METHOD PROTECTED OnExecute
VAR
    avgStrength : REAL;
END_VAR
hresult.Value := F_VN_LocateAxisAlignedEdges(
    ipSrcImage := ipSrcImage.Value,
    ipEdgePoints := ipEdgePoints.Value,
    aStartPoint := aStartPoint.Value,
    aEndPoint := aEndPoint.Value,
    nSearchWindowHeight := nSearchWindowHeight.Value,
    nKernelSize := nKernelSize.Value,
    nNumEdges := nNumEdges.Value,
    eEdgeSelection := eEdgeSelection.Value,
    fMinStrength := fMinStrength.Value,
    hrPrev := hrPrev.Value,
    fAvgStrength => avgStrength);

fAvgStrength.Value := avgStrength;
END_METHOD

METHOD PUBLIC PreExecutionCheck
VAR_INPUT
    Check : I_PreExecutionChecks;
END_VAR
Check.IsTrue(ipSrcImage.IsValid, 'ipSrcImage must contain an image');
Check.IsTrue(ipSrcImage.HasChannelCount(1), 'ipSrcImage must contain 1 channel');
Check.IsTrue((aStartPoint.Value[0] = aEndPoint.Value[0]) OR (aStartPoint.Value[1] = aEndPoint.Value[1]), 'aEndPoint must share the x- or y-coordinate of aStartPoint');
Check.IsTrue(nSearchWindowHeight.Value > 0, 'nSearchWindowHeight must be at least 1');
Check.IsTrue(nKernelSize.IsOdd, 'nKernelSize must be an odd number');
Check.IsTrue(nKernelSize.Value >= 3, 'nKernelSize must be at least 3');
Check.IsTrue(nNumEdges.Value > 0, 'nNumEdges must be at least 1');
END_METHOD

END_FUNCTION_BLOCK

// Nodes/Measurement/Node_F_VN_LocateAxisAlignedEdgesExp
{attribute 'linkalways'}
{attribute 'no_explicit_call' := 'This FB is a CLASS and must be accessed using methods or properties'}
{attribute 'enable_dynamic_creation'}
FUNCTION_BLOCK Node_F_VN_LocateAxisAlignedEdgesExp EXTENDS VisionNode
VAR
    ipSrcImage : _ITcVnImage;
    ipEdgePoints : _ITcVnContainer;
    aStartPoint : _TcVnPoint2_DINT;
    aEndPoint : _TcVnPoint2_DINT;
    nSearchWindowHeight : _UDINT(1);
    nKernelSize : _UDINT(5);
    nNumEdges : _UDINT(1);
    eEdgeSelection : _ETcVnEdgeSelection(ETcVnEdgeSelection.TCVN_ES_ANY);
    fMinStrength : _REAL(0.0);
    fSigma : _REAL(0.0);
    ipEdgeStrengths : _ITcVnContainer;
    ipDerivative : _ITcVnImage;
    hrPrev : _HRESULT(S_OK);
    fAvgStrength : _REAL(0.0);
    hresult : _HRESULT(S_OK);
END_VAR

METHOD FB_init : BOOL
VAR_INPUT
    bInitRetains : BOOL;
    bInCopyCode : BOOL;
END_VAR
AddInput('ipSrcImage', ipSrcImage);
AddOutput('ipEdgePoints', ipEdgePoints);
AddInput('aStartPoint', aStartPoint);
AddInput('aEndPoint', aEndPoint);
AddParameter('nSearchWindowHeight', nSearchWindowHeight);
AddParameter('nKernelSize', nKernelSize);
AddParameter('nNumEdges', nNumEdges);
AddParameter('eEdgeSelection', eEdgeSelection);
AddParameter('fMinStrength', fMinStrength);
AddParameter('fSigma', fSigma);
AddOutput('ipEdgeStrengths', ipEdgeStrengths);
AddOutput('ipDerivative', ipDerivative);
AddInput('hrPrev', hrPrev);
AddOutput('fAvgStrength', fAvgStrength);
AddOutput('hresult', hresult);
END_METHOD

METHOD PUBLIC Clone : I_Node
VAR
    pNode : POINTER TO Node_F_VN_LocateAxisAlignedEdgesExp;
END_VAR
pNode := __NEW(Node_F_VN_LocateAxisAlignedEdgesExp);
Clone := pNode^;
END_METHOD

METHOD PROTECTED OnExecute
VAR
    avgStrength : REAL;
END_VAR
hresult.Value := F_VN_LocateAxisAlignedEdgesExp(
    ipSrcImage := ipSrcImage.Value,
    ipEdgePoints := ipEdgePoints.Value,
    aStartPoint := aStartPoint.Value,
    aEndPoint := aEndPoint.Value,
    nSearchWindowHeight := nSearchWindowHeight.Value,
    nKernelSize := nKernelSize.Value,
    nNumEdges := nNumEdges.Value,
    eEdgeSelection := eEdgeSelection.Value,
    fMinStrength := fMinStrength.Value,
    fSigma := fSigma.Value,
    ipEdgeStrengths := ipEdgeStrengths.Value,
    ipDerivative := ipDerivative.Value,
    hrPrev := hrPrev.Value,
    fAvgStrength => avgStrength);

fAvgStrength.Value := avgStrength;
END_METHOD

METHOD PUBLIC PreExecutionCheck
VAR_INPUT
    Check : I_PreExecutionChecks;
END_VAR
Check.IsTrue(ipSrcImage.IsValid, 'ipSrcImage must contain an image');
Check.IsTrue(ipSrcImage.HasChannelCount(1), 'ipSrcImage must contain 1 channel');
Check.IsTrue((aStartPoint.Value[0] = aEndPoint.Value[0]) OR (aStartPoint.Value[1] = aEndPoint.Value[1]), 'aEndPoint must share the x- or y-coordinate of aStartPoint');
Check.IsTrue(nSearchWindowHeight.Value > 0, 'nSearchWindowHeight must be at least 1');
Check.IsTrue(nKernelSize.IsOdd, 'nKernelSize must be an odd number');
Check.IsTrue(nKernelSize.Value >= 3, 'nKernelSize must be at least 3');
Check.IsTrue(nNumEdges.Value > 0, 'nNumEdges must be at least 1');
// fSigma = 0 lets the function choose a value from nKernelSize.
Check.IsTrue(fSigma.Value >= 0.0, 'fSigma cannot be negative');
Check.IsTrue((ipDerivative.Value = 0) OR (ipDerivative.Value <> ipSrcImage.Value), 'ipDerivative must be different from the source image');
END_METHOD

END_FUNCTION_BLOCK

// Nodes/Measurement/Node_F_VN_LocateCircularArc
{attribute 'linkalways'} 
{attribute 'no_explicit_call' := 'This FB is a CLASS and must be accessed using methods or properties'}
{attribute 'enable_dynamic_creation'}
FUNCTION_BLOCK Node_F_VN_LocateCircularArc EXTENDS VisionNode
VAR
	ipSrcImage : _ITcVnImage;
	stCircularArc : _TcVnCircularArc;
	aCenter : _TcVnPoint2_REAL;
	fSearchRadius : _REAL(0.0);
	fArcDirectionRad : _LREAL(0.0);
	eEdgeDirection : _ETcVnEdgeDirection(ETcVnEdgeDirection.TCVN_ED_DARK_TO_LIGHT);
    fMinStrength : _REAL(0.0);
	hrPrev : _HRESULT(S_OK);
	hresult : _HRESULT(S_OK);
END_VAR

METHOD FB_init : BOOL
VAR_INPUT
	bInitRetains : BOOL; // if TRUE, the retain variables are initialized (warm start / cold start)
	bInCopyCode : BOOL;  // if TRUE, the instance afterwards gets moved into the copy code (online change)
END_VAR
AddInput('ipSrcImage', ipSrcImage);
AddInput('aCenter', aCenter);
AddInput('hrPrev', hrPrev);
AddParameter('fSearchRadius', fSearchRadius);
AddParameter('fArcDirectionRad', fArcDirectionRad);
AddParameter('eEdgeDirection', eEdgeDirection);
AddParameter('fMinStrength', fMinStrength);
AddOutput('stCircularArc', stCircularArc);
AddOutput('aCenter', aCenter);
AddOutput('hresult',hresult);
END_METHOD

METHOD PUBLIC  Clone : I_Node
VAR
	pNode : POINTER TO Node_F_VN_LocateCircularArc;
END_VAR
pNode := __NEW(Node_F_VN_LocateCircularArc);
Clone := pNode^;
END_METHOD

METHOD PROTECTED OnExecute
hresult.Value := F_VN_LocateCircularArc(
	ipSrcImage := ipSrcImage.Value,
	stCircularArc := stCircularArc.Value,
    aCenter := aCenter.Value,
    fSearchRadius := fSearchRadius.Value,
    fArcDirectionRad := fArcDirectionRad.Value,
	eEdgeDirection := eEdgeDirection.Value,
	fMinStrength := fMinStrength.Value,
	hrPrev := hrPrev.Value);
END_METHOD

METHOD PUBLIC PreExecutionCheck
VAR_INPUT
	Check : I_PreExecutionChecks;
END_VAR
VAR
	width : UDINT;
	height : UDINT;
	cx : REAL;
	cy : REAL;
END_VAR
// Source image (1 channel)
Check.IsTrue(ipSrcImage.IsValid, 'ipSrcImage must contain an image');
Check.IsTrue(ipSrcImage.HasChannelCount(1), 'ipSrcImage must contain 1 channel');
	
// Input search radius (starting FROM aCenter, should be greater than the actual circle radius but 
// aCenter + fSearchRadius should be within the image borders)
ipSrcImage.TryGetWidth(width);
ipSrcImage.TryGetHeight(height);

Check.IsTrue((width > 0), 'ipSrcImage have valid width');
Check.IsTrue((height > 0), 'ipSrcImage have valid height');
Check.IsTrue(fSearchRadius.Value > 0, 'fSearchRadius must be > 0');

cx := aCenter.Value[0];
cy := aCenter.Value[1];

Check.IsTrue(cx - fSearchRadius.Value >= 0, 'Search radius exceeds left border');
Check.IsTrue(cy - fSearchRadius.Value >= 0, 'Search radius exceeds top border');
Check.IsTrue(cx + fSearchRadius.Value < UDINT_TO_REAL(width), 'Search radius exceeds right border');
Check.IsTrue(cy + fSearchRadius.Value < UDINT_TO_REAL(height), 'Search radius exceeds bottom border');

// Input search starting direction in radian. Valid range is [-pi, +pi], where right is 0 rad, 
// top is -pi/2 rad and bottom +pi/2 rad. The circular arc should at least be valid in range 
// fArcDirectionRad +- 0.4 rad.
Check.IsTrue(fArcDirectionRad.Value >= -PI AND fArcDirectionRad.Value <= PI, 'fArcDirectionRad must be in [-pi, +pi]');
Check.IsTrue(fArcDirectionRad.Value - 0.4 >= -PI, 'fArcDirectionRad - 0.4 must be >= -pi');
Check.IsTrue(fArcDirectionRad.Value + 0.4 <=  PI, 'fArcDirectionRad + 0.4 must be <= +pi');
END_METHOD

END_FUNCTION_BLOCK

// Nodes/Measurement/Node_F_VN_LocateCircularArcExp
{attribute 'linkalways'}
{attribute 'no_explicit_call' := 'This FB is a CLASS and must be accessed using methods or properties'}
{attribute 'enable_dynamic_creation'}
FUNCTION_BLOCK Node_F_VN_LocateCircularArcExp EXTENDS VisionNode
VAR
    ipSrcImage : _ITcVnImage;
    stCircularArc : _TcVnCircularArc;
    aCenter : _TcVnPoint2_REAL;
    fSearchRadius : _REAL(0.0);
    fArcDirectionRad : _LREAL(0.0);
    eEdgeDirection : _ETcVnEdgeDirection(ETcVnEdgeDirection.TCVN_ED_DARK_TO_LIGHT);
    fMinStrength : _REAL(0.0);
    fAngleStepRad : _LREAL(0.1);
    nMaxThickness : _UDINT(10);
    bInvertSearchDirection : _BOOL(FALSE);
    nSubpixelsIterations : _UDINT(10);
    fApproxPrecision : _REAL(0.001);
    eAlgorithm : _ETcVnEdgeDetectionAlgorithm(ETcVnEdgeDetectionAlgorithm.TCVN_EDA_INTERPOLATION);
    ipContourPoints : _ITcVnContainer;
    hrPrev : _HRESULT(S_OK);
    hresult : _HRESULT(S_OK);
END_VAR

METHOD FB_init : BOOL
VAR_INPUT
    bInitRetains : BOOL;
    bInCopyCode : BOOL;
END_VAR
AddInput('ipSrcImage', ipSrcImage);
AddOutput('stCircularArc', stCircularArc);
AddInput('aCenter', aCenter);
AddParameter('fSearchRadius', fSearchRadius);
AddParameter('fArcDirectionRad', fArcDirectionRad);
AddParameter('eEdgeDirection', eEdgeDirection);
AddParameter('fMinStrength', fMinStrength);
AddParameter('fAngleStepRad', fAngleStepRad);
AddParameter('nMaxThickness', nMaxThickness);
AddParameter('bInvertSearchDirection', bInvertSearchDirection);
AddParameter('nSubpixelsIterations', nSubpixelsIterations);
AddParameter('fApproxPrecision', fApproxPrecision);
AddParameter('eAlgorithm', eAlgorithm);
AddOutput('ipContourPoints', ipContourPoints);
AddInput('hrPrev', hrPrev);
AddOutput('aCenter', aCenter);
AddOutput('hresult', hresult);
END_METHOD

METHOD PUBLIC Clone : I_Node
VAR
    pNode : POINTER TO Node_F_VN_LocateCircularArcExp;
END_VAR
pNode := __NEW(Node_F_VN_LocateCircularArcExp);
Clone := pNode^;
END_METHOD

METHOD PROTECTED OnExecute
hresult.Value := F_VN_LocateCircularArcExp(
    ipSrcImage := ipSrcImage.Value,
    stCircularArc := stCircularArc.Value,
    aCenter := aCenter.Value,
    fSearchRadius := fSearchRadius.Value,
    fArcDirectionRad := fArcDirectionRad.Value,
    eEdgeDirection := eEdgeDirection.Value,
    fMinStrength := fMinStrength.Value,
    fAngleStepRad := fAngleStepRad.Value,
    nMaxThickness := nMaxThickness.Value,
    bInvertSearchDirection := bInvertSearchDirection.Value,
    nSubpixelsIterations := nSubpixelsIterations.Value,
    fApproxPrecision := fApproxPrecision.Value,
    eAlgorithm := eAlgorithm.Value,
    ipContourPoints := ipContourPoints.Value,
    hrPrev := hrPrev.Value);
END_METHOD

METHOD PUBLIC PreExecutionCheck
VAR_INPUT
    Check : I_PreExecutionChecks;
END_VAR
VAR
    width : UDINT;
    height : UDINT;
    cx : REAL;
    cy : REAL;
END_VAR
Check.IsTrue(ipSrcImage.IsValid, 'ipSrcImage must contain an image');
Check.IsTrue(ipSrcImage.HasChannelCount(1), 'ipSrcImage must contain 1 channel');

// Input search radius (starting FROM aCenter, should be greater than the actual radius but
// aCenter + fSearchRadius should be within the image borders)
ipSrcImage.TryGetWidth(width);
ipSrcImage.TryGetHeight(height);

Check.IsTrue((width > 0), 'ipSrcImage have valid width');
Check.IsTrue((height > 0), 'ipSrcImage have valid height');
Check.IsTrue(fSearchRadius.Value > 0, 'fSearchRadius must be > 0');

cx := aCenter.Value[0];
cy := aCenter.Value[1];

Check.IsTrue(cx - fSearchRadius.Value >= 0, 'Search radius exceeds left border');
Check.IsTrue(cy - fSearchRadius.Value >= 0, 'Search radius exceeds top border');
Check.IsTrue(cx + fSearchRadius.Value < UDINT_TO_REAL(width), 'Search radius exceeds right border');
Check.IsTrue(cy + fSearchRadius.Value < UDINT_TO_REAL(height), 'Search radius exceeds bottom border');

// Input search starting direction in radian. Valid range is [-pi, +pi], where right is 0 rad,
// top is -pi/2 rad and bottom +pi/2 rad. The circular arc should at least be valid in range
// fArcDirectionRad +- 4 * fAngleStepRad.
Check.IsTrue(fAngleStepRad.Value > 0.0, 'fAngleStepRad must be greater than 0');
Check.IsTrue(fArcDirectionRad.Value >= -PI AND fArcDirectionRad.Value <= PI, 'fArcDirectionRad must be in [-pi, +pi]');
Check.IsTrue(fArcDirectionRad.Value - 4.0 * fAngleStepRad.Value >= -PI, 'fArcDirectionRad - 4 * fAngleStepRad must be >= -pi');
Check.IsTrue(fArcDirectionRad.Value + 4.0 * fAngleStepRad.Value <=  PI, 'fArcDirectionRad + 4 * fAngleStepRad must be <= +pi');

Check.IsTrue(nMaxThickness.Value > 0, 'nMaxThickness must be at least 1');
Check.IsTrue(nSubpixelsIterations.Value > 0, 'nSubpixelsIterations must be greater than 0');
Check.IsTrue((eAlgorithm.Value = ETcVnEdgeDetectionAlgorithm.TCVN_EDA_INTERPOLATION) OR
             (fApproxPrecision.Value > 0.0), 'fApproxPrecision must be greater than 0 for the approximation algorithms');
END_METHOD

END_FUNCTION_BLOCK

// Nodes/Measurement/Node_F_VN_LocateCircularArcExp2
{attribute 'linkalways'}
{attribute 'no_explicit_call' := 'This FB is a CLASS and must be accessed using methods or properties'}
{attribute 'enable_dynamic_creation'}
FUNCTION_BLOCK Node_F_VN_LocateCircularArcExp2 EXTENDS VisionNode
VAR
    ipSrcImage : _ITcVnImage;
    stCircularArc : _TcVnCircularArc;
    aCenter : _TcVnPoint2_REAL;
    fSearchRadius : _REAL(0.0);
    fArcDirectionRad : _LREAL(0.0);
    eEdgeDirection : _ETcVnEdgeDirection(ETcVnEdgeDirection.TCVN_ED_DARK_TO_LIGHT);
    fMinStrength : _REAL(0.0);
    fAngleStepRad : _LREAL(0.1);
    nMaxThickness : _UDINT(10);
    bInvertSearchDirection : _BOOL(FALSE);
    nSubpixelsIterations : _UDINT(10);
    fApproxPrecision : _REAL(0.001);
    eAlgorithm : _ETcVnEdgeDetectionAlgorithm(ETcVnEdgeDetectionAlgorithm.TCVN_EDA_INTERPOLATION);
    ipContourPoints : _ITcVnContainer;
    fRangeCutoffFactor : _REAL(0.135);
    hrPrev : _HRESULT(S_OK);
    hresult : _HRESULT(S_OK);
END_VAR

METHOD FB_init : BOOL
VAR_INPUT
    bInitRetains : BOOL;
    bInCopyCode : BOOL;
END_VAR
AddInput('ipSrcImage', ipSrcImage);
AddOutput('stCircularArc', stCircularArc);
AddInput('aCenter', aCenter);
AddParameter('fSearchRadius', fSearchRadius);
AddParameter('fArcDirectionRad', fArcDirectionRad);
AddParameter('eEdgeDirection', eEdgeDirection);
AddParameter('fMinStrength', fMinStrength);
AddParameter('fAngleStepRad', fAngleStepRad);
AddParameter('nMaxThickness', nMaxThickness);
AddParameter('bInvertSearchDirection', bInvertSearchDirection);
AddParameter('nSubpixelsIterations', nSubpixelsIterations);
AddParameter('fApproxPrecision', fApproxPrecision);
AddParameter('eAlgorithm', eAlgorithm);
AddOutput('ipContourPoints', ipContourPoints);
AddParameter('fRangeCutoffFactor', fRangeCutoffFactor);
AddInput('hrPrev', hrPrev);
AddOutput('aCenter', aCenter);
AddOutput('hresult', hresult);
END_METHOD

METHOD PUBLIC Clone : I_Node
VAR
    pNode : POINTER TO Node_F_VN_LocateCircularArcExp2;
END_VAR
pNode := __NEW(Node_F_VN_LocateCircularArcExp2);
Clone := pNode^;
END_METHOD

METHOD PROTECTED OnExecute
hresult.Value := F_VN_LocateCircularArcExp2(
    ipSrcImage := ipSrcImage.Value,
    stCircularArc := stCircularArc.Value,
    aCenter := aCenter.Value,
    fSearchRadius := fSearchRadius.Value,
    fArcDirectionRad := fArcDirectionRad.Value,
    eEdgeDirection := eEdgeDirection.Value,
    fMinStrength := fMinStrength.Value,
    fAngleStepRad := fAngleStepRad.Value,
    nMaxThickness := nMaxThickness.Value,
    bInvertSearchDirection := bInvertSearchDirection.Value,
    nSubpixelsIterations := nSubpixelsIterations.Value,
    fApproxPrecision := fApproxPrecision.Value,
    eAlgorithm := eAlgorithm.Value,
    ipContourPoints := ipContourPoints.Value,
    fRangeCutoffFactor := fRangeCutoffFactor.Value,
    hrPrev := hrPrev.Value);
END_METHOD

METHOD PUBLIC PreExecutionCheck
VAR_INPUT
    Check : I_PreExecutionChecks;
END_VAR
VAR
    width : UDINT;
    height : UDINT;
    cx : REAL;
    cy : REAL;
END_VAR
Check.IsTrue(ipSrcImage.IsValid, 'ipSrcImage must contain an image');
Check.IsTrue(ipSrcImage.HasChannelCount(1), 'ipSrcImage must contain 1 channel');

// Input search radius (starting FROM aCenter, should be greater than the actual radius but
// aCenter + fSearchRadius should be within the image borders)
ipSrcImage.TryGetWidth(width);
ipSrcImage.TryGetHeight(height);

Check.IsTrue((width > 0), 'ipSrcImage have valid width');
Check.IsTrue((height > 0), 'ipSrcImage have valid height');
Check.IsTrue(fSearchRadius.Value > 0, 'fSearchRadius must be > 0');

cx := aCenter.Value[0];
cy := aCenter.Value[1];

Check.IsTrue(cx - fSearchRadius.Value >= 0, 'Search radius exceeds left border');
Check.IsTrue(cy - fSearchRadius.Value >= 0, 'Search radius exceeds top border');
Check.IsTrue(cx + fSearchRadius.Value < UDINT_TO_REAL(width), 'Search radius exceeds right border');
Check.IsTrue(cy + fSearchRadius.Value < UDINT_TO_REAL(height), 'Search radius exceeds bottom border');

// Input search starting direction in radian. Valid range is [-pi, +pi], where right is 0 rad,
// top is -pi/2 rad and bottom +pi/2 rad. The circular arc should at least be valid in range
// fArcDirectionRad +- 4 * fAngleStepRad.
Check.IsTrue(fAngleStepRad.Value > 0.0, 'fAngleStepRad must be greater than 0');
Check.IsTrue(fArcDirectionRad.Value >= -PI AND fArcDirectionRad.Value <= PI, 'fArcDirectionRad must be in [-pi, +pi]');
Check.IsTrue(fArcDirectionRad.Value - 4.0 * fAngleStepRad.Value >= -PI, 'fArcDirectionRad - 4 * fAngleStepRad must be >= -pi');
Check.IsTrue(fArcDirectionRad.Value + 4.0 * fAngleStepRad.Value <=  PI, 'fArcDirectionRad + 4 * fAngleStepRad must be <= +pi');

Check.IsTrue(nMaxThickness.Value > 0, 'nMaxThickness must be at least 1');
Check.IsTrue(nSubpixelsIterations.Value > 0, 'nSubpixelsIterations must be greater than 0');
Check.IsTrue((eAlgorithm.Value = ETcVnEdgeDetectionAlgorithm.TCVN_EDA_INTERPOLATION) OR
             (fApproxPrecision.Value > 0.0), 'fApproxPrecision must be greater than 0 for the approximation algorithms');
END_METHOD

END_FUNCTION_BLOCK

// Nodes/Measurement/Node_F_VN_LocateEdge
{attribute 'linkalways'} 
{attribute 'no_explicit_call' := 'This FB is a CLASS and must be accessed using methods or properties'}
{attribute 'enable_dynamic_creation'}
FUNCTION_BLOCK Node_F_VN_LocateEdge EXTENDS VisionNode
VAR
	ipSrcImage : _ITcVnImage;
    ipEdgePoints : _ITcVnContainer;
    aStartPoint : _TcVnPoint2_REAL;
    aEndPoint : _TcVnPoint2_REAL;
	eEdgeDirection : _ETcVnEdgeDirection(ETcVnEdgeDirection.TCVN_ED_DARK_TO_LIGHT);
    fMinStrength : _REAL(0.0);
    nSearchLines : _UDINT(1);
    hrPrev : _HRESULT(S_OK);
    fAvgStrength : _REAL(0.0);
	hresult : _HRESULT(S_OK);
END_VAR

METHOD FB_init : BOOL
VAR_INPUT
	bInitRetains : BOOL; // if TRUE, the retain variables are initialized (warm start / cold start)
	bInCopyCode : BOOL;  // if TRUE, the instance afterwards gets moved into the copy code (online change)
END_VAR
AddInput('ipSrcImage', ipSrcImage);
AddInput('aStartPoint', aStartPoint);
AddInput('aEndPoint', aEndPoint);
AddParameter('eEdgeDirection', eEdgeDirection);
AddParameter('fMinStrength', fMinStrength);
AddParameter('nSearchLines', nSearchLines);
AddInput('hrPrev', hrPrev);
AddOutput('ipEdgePoints', ipEdgePoints);
AddOutput('fAvgStrength', fAvgStrength);
AddOutput('hresult',hresult);
END_METHOD

METHOD PUBLIC  Clone : I_Node
VAR
	pNode : POINTER TO Node_F_VN_LocateEdge;
END_VAR
pNode := __NEW(Node_F_VN_LocateEdge);
Clone := pNode^;
END_METHOD

METHOD PROTECTED OnExecute
VAR
    avgStrength : REAL;
END_VAR
hresult.Value := F_VN_LocateEdge(
	ipSrcImage := ipSrcImage.Value,
	ipEdgePoints := ipEdgePoints.Value,
    aStartPoint := aStartPoint.Value,
    aEndPoint := aEndPoint.Value,
    eEdgeDirection := eEdgeDirection.Value,
	fMinStrength := fMinStrength.Value,
	nSearchLines := nSearchLines.Value,
	hrPrev := hrPrev.Value,
    fAvgStrength => avgStrength);
    
fAvgStrength.Value := avgStrength;
END_METHOD

METHOD PUBLIC PreExecutionCheck
VAR_INPUT
	Check : I_PreExecutionChecks;
END_VAR
Check.IsTrue(ipSrcImage.IsValid, 'ipSrcImage must contain an image');
Check.IsTrue(ipSrcImage.HasChannelCount(1), 'ipSrcImage must contain 1 channel');
Check.IsTrue(nSearchLines.IsOdd, 'nSearchLines must be an odd number');
END_METHOD

END_FUNCTION_BLOCK

// Nodes/Measurement/Node_F_VN_LocateEdgeExp
{attribute 'linkalways'} 
{attribute 'no_explicit_call' := 'This FB is a CLASS and must be accessed using methods or properties'}
{attribute 'enable_dynamic_creation'}
FUNCTION_BLOCK Node_F_VN_LocateEdgeExp EXTENDS VisionNode
VAR
	ipSrcImage : _ITcVnImage;
    ipEdgePoints : _ITcVnContainer;
    aStartPoint : _TcVnPoint2_REAL;
    aEndPoint : _TcVnPoint2_REAL;
	eEdgeDirection : _ETcVnEdgeDirection(ETcVnEdgeDirection.TCVN_ED_DARK_TO_LIGHT);
    fMinStrength : _REAL(0.0);
    nSearchLines : _UDINT(1);
    fSearchLineDist : _REAL(0.0);
    nMaxThickness : _UDINT(0);
    nSubpixelsIterations : _UDINT(0);
    fApproxPrecision : _REAL(0.0);
    eAlgorithm : _ETcVnEdgeDetectionAlgorithm(ETcVnEdgeDetectionAlgorithm.TCVN_EDA_INTERPOLATION);
    hrPrev : _HRESULT(S_OK);
    fAvgStrength : _REAL(0.0);
	hresult : _HRESULT(S_OK);
END_VAR

METHOD FB_init : BOOL
VAR_INPUT
	bInitRetains : BOOL; // if TRUE, the retain variables are initialized (warm start / cold start)
	bInCopyCode : BOOL;  // if TRUE, the instance afterwards gets moved into the copy code (online change)
END_VAR
AddInput('ipSrcImage', ipSrcImage);
AddInput('aStartPoint', aStartPoint);
AddInput('aEndPoint', aEndPoint);
AddParameter('eEdgeDirection', eEdgeDirection);
AddParameter('fMinStrength', fMinStrength);
AddParameter('nSearchLines', nSearchLines);
AddParameter('fSearchLineDist', fSearchLineDist);
AddParameter('nMaxThickness', nMaxThickness);
AddParameter('nSubpixelsIterations', nSubpixelsIterations);
AddParameter('fApproxPrecision', fApproxPrecision);
AddParameter('eAlgorithm', eAlgorithm);
AddInput('hrPrev', hrPrev);
AddOutput('ipEdgePoints', ipEdgePoints);
AddOutput('fAvgStrength', fAvgStrength);
AddOutput('hresult',hresult);
END_METHOD

METHOD PUBLIC  Clone : I_Node
VAR
	pNode : POINTER TO Node_F_VN_LocateEdgeExp;
END_VAR
pNode := __NEW(Node_F_VN_LocateEdgeExp);
Clone := pNode^;
END_METHOD

METHOD PROTECTED OnExecute
VAR
    avgStrength : REAL;
END_VAR
hresult.Value := F_VN_LocateEdgeExp(
	ipSrcImage := ipSrcImage.Value,
	ipEdgePoints := ipEdgePoints.Value,
    aStartPoint := aStartPoint.Value,
    aEndPoint := aEndPoint.Value,
    eEdgeDirection := eEdgeDirection.Value,
	fMinStrength := fMinStrength.Value,
	nSearchLines := nSearchLines.Value,
    fSearchLineDist := fSearchLineDist.Value,
    nMaxThickness := nMaxThickness.Value,
    nSubpixelsIterations := nSubpixelsIterations.Value,
    fApproxPrecision := fApproxPrecision.Value,
    eAlgorithm := eAlgorithm.Value,
	hrPrev:= hrPrev.Value,
    fAvgStrength => avgStrength);
    
fAvgStrength.Value := avgStrength;
END_METHOD

METHOD PUBLIC PreExecutionCheck
VAR_INPUT
	Check : I_PreExecutionChecks;
END_VAR
Check.IsTrue(ipSrcImage.IsValid, 'ipSrcImage must contain an image');
Check.IsTrue(ipSrcImage.HasChannelCount(1), 'ipSrcImage must contain 1 channel');
Check.IsTrue(nSearchLines.IsOdd, 'nSearchLines must be an odd number');
Check.IsTrue((fSearchLineDist.Value > 0.0), 'nSearchLineDist must be greater than 0');
END_METHOD

END_FUNCTION_BLOCK

// Nodes/Measurement/Node_F_VN_LocateEdgeExp2
{attribute 'linkalways'}
{attribute 'no_explicit_call' := 'This FB is a CLASS and must be accessed using methods or properties'}
{attribute 'enable_dynamic_creation'}
FUNCTION_BLOCK Node_F_VN_LocateEdgeExp2 EXTENDS VisionNode
VAR
    ipSrcImage : _ITcVnImage;
    ipEdgePoints : _ITcVnContainer;
    aStartPoint : _TcVnPoint2_REAL;
    aEndPoint : _TcVnPoint2_REAL;
    eEdgeDirection : _ETcVnEdgeDirection(ETcVnEdgeDirection.TCVN_ED_DARK_TO_LIGHT);
    fMinStrength : _REAL(0.0);
    nSearchLines : _UDINT(1);
    fSearchLineDist : _REAL(1.0);
    nMaxThickness : _UDINT(10);
    nSubpixelsIterations : _UDINT(10);
    fApproxPrecision : _REAL(0.001);
    eAlgorithm : _ETcVnEdgeDetectionAlgorithm(ETcVnEdgeDetectionAlgorithm.TCVN_EDA_INTERPOLATION);
    fRangeCutoffFactor : _REAL(0.135);
    ipEdgeStrengths : _ITcVnContainer;
    hrPrev : _HRESULT(S_OK);
    fAvgStrength : _REAL(0.0);
    hresult : _HRESULT(S_OK);
END_VAR

METHOD FB_init : BOOL
VAR_INPUT
    bInitRetains : BOOL;
    bInCopyCode : BOOL;
END_VAR
AddInput('ipSrcImage', ipSrcImage);
AddOutput('ipEdgePoints', ipEdgePoints);
AddInput('aStartPoint', aStartPoint);
AddInput('aEndPoint', aEndPoint);
AddParameter('eEdgeDirection', eEdgeDirection);
AddParameter('fMinStrength', fMinStrength);
AddParameter('nSearchLines', nSearchLines);
AddParameter('fSearchLineDist', fSearchLineDist);
AddParameter('nMaxThickness', nMaxThickness);
AddParameter('nSubpixelsIterations', nSubpixelsIterations);
AddParameter('fApproxPrecision', fApproxPrecision);
AddParameter('eAlgorithm', eAlgorithm);
AddParameter('fRangeCutoffFactor', fRangeCutoffFactor);
AddOutput('ipEdgeStrengths', ipEdgeStrengths);
AddInput('hrPrev', hrPrev);
AddOutput('fAvgStrength', fAvgStrength);
AddOutput('hresult', hresult);
END_METHOD

METHOD PUBLIC Clone : I_Node
VAR
    pNode : POINTER TO Node_F_VN_LocateEdgeExp2;
END_VAR
pNode := __NEW(Node_F_VN_LocateEdgeExp2);
Clone := pNode^;
END_METHOD

METHOD PROTECTED OnExecute
VAR
    avgStrength : REAL;
END_VAR
hresult.Value := F_VN_LocateEdgeExp2(
    ipSrcImage := ipSrcImage.Value,
    ipEdgePoints := ipEdgePoints.Value,
    aStartPoint := aStartPoint.Value,
    aEndPoint := aEndPoint.Value,
    eEdgeDirection := eEdgeDirection.Value,
    fMinStrength := fMinStrength.Value,
    nSearchLines := nSearchLines.Value,
    fSearchLineDist := fSearchLineDist.Value,
    nMaxThickness := nMaxThickness.Value,
    nSubpixelsIterations := nSubpixelsIterations.Value,
    fApproxPrecision := fApproxPrecision.Value,
    eAlgorithm := eAlgorithm.Value,
    fRangeCutoffFactor := fRangeCutoffFactor.Value,
    ipEdgeStrengths := ipEdgeStrengths.Value,
    hrPrev := hrPrev.Value,
    fAvgStrength => avgStrength);

fAvgStrength.Value := avgStrength;
END_METHOD

METHOD PUBLIC PreExecutionCheck
VAR_INPUT
    Check : I_PreExecutionChecks;
END_VAR
Check.IsTrue(ipSrcImage.IsValid, 'ipSrcImage must contain an image');
Check.IsTrue(ipSrcImage.HasChannelCount(1), 'ipSrcImage must contain 1 channel');
Check.IsTrue(nSearchLines.IsOdd, 'nSearchLines must be an odd number');
Check.IsTrue(fSearchLineDist.Value > 0.0, 'fSearchLineDist must be greater than 0');
Check.IsTrue(nMaxThickness.Value > 0, 'nMaxThickness must be at least 1');
Check.IsTrue(nSubpixelsIterations.Value > 0, 'nSubpixelsIterations must be greater than 0');
Check.IsTrue((eAlgorithm.Value = ETcVnEdgeDetectionAlgorithm.TCVN_EDA_INTERPOLATION) OR
             (fApproxPrecision.Value > 0.0), 'fApproxPrecision must be greater than 0 for the approximation algorithms');
END_METHOD

END_FUNCTION_BLOCK

// Nodes/Measurement/Node_F_VN_LocateEdges
{attribute 'linkalways'} 
{attribute 'no_explicit_call' := 'This FB is a CLASS and must be accessed using methods or properties'}
{attribute 'enable_dynamic_creation'}
FUNCTION_BLOCK Node_F_VN_LocateEdges EXTENDS VisionNode
VAR
	ipSrcImage : _ITcVnImage;
    ipEdgePoints : _ITcVnContainer;
    aStartPoint : _TcVnPoint2_REAL;
    aEndPoint : _TcVnPoint2_REAL;
    nNumEdges : _UDINT(0);
	eEdgeDirection : _ETcVnEdgeDirection(ETcVnEdgeDirection.TCVN_ED_DARK_TO_LIGHT);
    bAlternateDirection : _BOOL(FALSE);
    fMinStrength : _REAL(0.0);
    nSearchLines : _UDINT(1);
    hrPrev : _HRESULT(S_OK);
    fAvgStrength : _REAL(0.0);
	hresult : _HRESULT(S_OK);
END_VAR

METHOD FB_init : BOOL
VAR_INPUT
	bInitRetains : BOOL; // if TRUE, the retain variables are initialized (warm start / cold start)
	bInCopyCode : BOOL;  // if TRUE, the instance afterwards gets moved into the copy code (online change)
END_VAR
AddInput('ipSrcImage', ipSrcImage);
AddInput('aStartPoint', aStartPoint);
AddInput('aEndPoint', aEndPoint);
AddParameter('nNumEdges', nNumEdges);
AddParameter('eEdgeDirection', eEdgeDirection);
AddParameter('bAlternateDirection', bAlternateDirection);
AddParameter('fMinStrength', fMinStrength);
AddParameter('nSearchLines', nSearchLines);
AddInput('hrPrev', hrPrev);
AddOutput('ipEdgePoints', ipEdgePoints);
AddOutput('fAvgStrength', fAvgStrength);
AddOutput('hresult',hresult);
END_METHOD

METHOD PUBLIC  Clone : I_Node
VAR
	pNode : POINTER TO Node_F_VN_LocateEdges;
END_VAR
pNode := __NEW(Node_F_VN_LocateEdges);
Clone := pNode^;
END_METHOD

METHOD PROTECTED OnExecute
VAR
    avgStrength : REAL;
END_VAR
hresult.Value := F_VN_LocateEdges(
	ipSrcImage := ipSrcImage.Value,
	ipEdgePoints := ipEdgePoints.Value,
    aStartPoint := aStartPoint.Value,
    aEndPoint := aEndPoint.Value,
    nNumEdges := nNumEdges.Value,
    eEdgeDirection := eEdgeDirection.Value,
    bAlternateDirection := bAlternateDirection.Value,
	fMinStrength := fMinStrength.Value,
	nSearchLines := nSearchLines.Value,
	hrPrev := hrPrev.Value,
    fAvgStrength => avgStrength);
    
fAvgStrength.Value := avgStrength;
END_METHOD

METHOD PUBLIC PreExecutionCheck
VAR_INPUT
	Check : I_PreExecutionChecks;
END_VAR
Check.IsTrue(ipSrcImage.IsValid, 'ipSrcImage must contain an image');
Check.IsTrue(ipSrcImage.HasChannelCount(1), 'ipSrcImage must contain 1 channel');
Check.IsTrue(nSearchLines.IsOdd, 'nSearchLines must be an odd number');
END_METHOD

END_FUNCTION_BLOCK

// Nodes/Measurement/Node_F_VN_LocateEdgesExp
{attribute 'linkalways'} 
{attribute 'no_explicit_call' := 'This FB is a CLASS and must be accessed using methods or properties'}
{attribute 'enable_dynamic_creation'}
FUNCTION_BLOCK Node_F_VN_LocateEdgesExp EXTENDS VisionNode
VAR
	ipSrcImage : _ITcVnImage;
    ipEdgePoints : _ITcVnContainer;
    aStartPoint : _TcVnPoint2_REAL;
    aEndPoint : _TcVnPoint2_REAL;
    nNumEdges : _UDINT(0);
	eEdgeDirection : _ETcVnEdgeDirection(ETcVnEdgeDirection.TCVN_ED_DARK_TO_LIGHT);
    bAlternateDirection : _BOOL(FALSE);
    fMinStrength : _REAL(0.0);
    nSearchLines : _UDINT(1);
    fSearchLineDist : _REAL(0.0);
    nMaxThickness : _UDINT(0);
    nSubpixelsIterations : _UDINT(0);
    fApproxPrecision : _REAL(0.0);
    eAlgorithm : _ETcVnEdgeDetectionAlgorithm(ETcVnEdgeDetectionAlgorithm.TCVN_EDA_INTERPOLATION);
    hrPrev : _HRESULT(S_OK);
    fAvgStrength : _REAL(0.0);
	hresult : _HRESULT(S_OK);
END_VAR

METHOD FB_init : BOOL
VAR_INPUT
	bInitRetains : BOOL; // if TRUE, the retain variables are initialized (warm start / cold start)
	bInCopyCode : BOOL;  // if TRUE, the instance afterwards gets moved into the copy code (online change)
END_VAR
AddInput('ipSrcImage', ipSrcImage);
AddInput('aStartPoint', aStartPoint);
AddInput('aEndPoint', aEndPoint);
AddParameter('nNumEdges', nNumEdges);
AddParameter('eEdgeDirection', eEdgeDirection);
AddParameter('bAlternateDirection', bAlternateDirection);
AddParameter('fMinStrength', fMinStrength);
AddParameter('nSearchLines', nSearchLines);
AddParameter('fSearchLineDist', fSearchLineDist);
AddParameter('nMaxThickness', nMaxThickness);
AddParameter('nSubpixelsIterations', nSubpixelsIterations);
AddParameter('fApproxPrecision', fApproxPrecision);
AddParameter('eAlgorithm', eAlgorithm);
AddInput('hrPrev', hrPrev);
AddOutput('ipEdgePoints', ipEdgePoints);
AddOutput('fAvgStrength', fAvgStrength);
AddOutput('hresult',hresult);
END_METHOD

METHOD PUBLIC  Clone : I_Node
VAR
	pNode : POINTER TO Node_F_VN_LocateEdgesExp;
END_VAR
pNode := __NEW(Node_F_VN_LocateEdgesExp);
Clone := pNode^;
END_METHOD

METHOD PROTECTED OnExecute
VAR
    avgStrength : REAL;
END_VAR
hresult.Value := F_VN_LocateEdgesExp(
	ipSrcImage := ipSrcImage.Value,
	ipEdgePoints := ipEdgePoints.Value,
    aStartPoint := aStartPoint.Value,
    aEndPoint := aEndPoint.Value,
    nNumEdges := nNumEdges.Value,
    eEdgeDirection := eEdgeDirection.Value,
    bAlternateDirection := bAlternateDirection.Value,
	fMinStrength := fMinStrength.Value,
	nSearchLines := nSearchLines.Value,
    fSearchLineDist := fSearchLineDist.Value,
    nMaxThickness := nMaxThickness.Value,
    nSubpixelsIterations := nSubpixelsIterations.Value,
    fApproxPrecision := fApproxPrecision.Value,
    eAlgorithm := eAlgorithm.Value,
	hrPrev := hrPrev.Value,
    fAvgStrength => avgStrength);
    
fAvgStrength.Value := avgStrength;
END_METHOD

METHOD PUBLIC PreExecutionCheck
VAR_INPUT
	Check : I_PreExecutionChecks;
END_VAR
Check.IsTrue(ipSrcImage.IsValid, 'ipSrcImage must contain an image');
Check.IsTrue(ipSrcImage.HasChannelCount(1), 'ipSrcImage must contain 1 channel');
Check.IsTrue(nSearchLines.IsOdd, 'nSearchLines must be an odd number');
Check.IsTrue((fSearchLineDist.Value > 0.0), 'nSearchLineDist must be greater than 0');
END_METHOD

END_FUNCTION_BLOCK

// Nodes/Measurement/Node_F_VN_LocateEdgesExp2
{attribute 'linkalways'}
{attribute 'no_explicit_call' := 'This FB is a CLASS and must be accessed using methods or properties'}
{attribute 'enable_dynamic_creation'}
FUNCTION_BLOCK Node_F_VN_LocateEdgesExp2 EXTENDS VisionNode
VAR
    ipSrcImage : _ITcVnImage;
    ipEdgePoints : _ITcVnContainer;
    aStartPoint : _TcVnPoint2_REAL;
    aEndPoint : _TcVnPoint2_REAL;
    nNumEdges : _UDINT(1);
    eEdgeDirection : _ETcVnEdgeDirection(ETcVnEdgeDirection.TCVN_ED_DARK_TO_LIGHT);
    bAlternateDirection : _BOOL(FALSE);
    fMinStrength : _REAL(0.0);
    nSearchLines : _UDINT(1);
    fSearchLineDist : _REAL(1.0);
    nMaxThickness : _UDINT(10);
    nSubpixelsIterations : _UDINT(10);
    fApproxPrecision : _REAL(0.001);
    eAlgorithm : _ETcVnEdgeDetectionAlgorithm(ETcVnEdgeDetectionAlgorithm.TCVN_EDA_INTERPOLATION);
    fRangeCutoffFactor : _REAL(0.135);
    ipEdgeStrengths : _ITcVnContainer;
    bAvgEdgeStrengths : _BOOL(FALSE);
    hrPrev : _HRESULT(S_OK);
    fAvgStrength : _REAL(0.0);
    hresult : _HRESULT(S_OK);
END_VAR

METHOD FB_init : BOOL
VAR_INPUT
    bInitRetains : BOOL;
    bInCopyCode : BOOL;
END_VAR
AddInput('ipSrcImage', ipSrcImage);
AddOutput('ipEdgePoints', ipEdgePoints);
AddInput('aStartPoint', aStartPoint);
AddInput('aEndPoint', aEndPoint);
AddParameter('nNumEdges', nNumEdges);
AddParameter('eEdgeDirection', eEdgeDirection);
AddParameter('bAlternateDirection', bAlternateDirection);
AddParameter('fMinStrength', fMinStrength);
AddParameter('nSearchLines', nSearchLines);
AddParameter('fSearchLineDist', fSearchLineDist);
AddParameter('nMaxThickness', nMaxThickness);
AddParameter('nSubpixelsIterations', nSubpixelsIterations);
AddParameter('fApproxPrecision', fApproxPrecision);
AddParameter('eAlgorithm', eAlgorithm);
AddParameter('fRangeCutoffFactor', fRangeCutoffFactor);
AddOutput('ipEdgeStrengths', ipEdgeStrengths);
AddParameter('bAvgEdgeStrengths', bAvgEdgeStrengths);
AddInput('hrPrev', hrPrev);
AddOutput('fAvgStrength', fAvgStrength);
AddOutput('hresult', hresult);
END_METHOD

METHOD PUBLIC Clone : I_Node
VAR
    pNode : POINTER TO Node_F_VN_LocateEdgesExp2;
END_VAR
pNode := __NEW(Node_F_VN_LocateEdgesExp2);
Clone := pNode^;
END_METHOD

METHOD PROTECTED OnExecute
VAR
    avgStrength : REAL;
END_VAR
hresult.Value := F_VN_LocateEdgesExp2(
    ipSrcImage := ipSrcImage.Value,
    ipEdgePoints := ipEdgePoints.Value,
    aStartPoint := aStartPoint.Value,
    aEndPoint := aEndPoint.Value,
    nNumEdges := nNumEdges.Value,
    eEdgeDirection := eEdgeDirection.Value,
    bAlternateDirection := bAlternateDirection.Value,
    fMinStrength := fMinStrength.Value,
    nSearchLines := nSearchLines.Value,
    fSearchLineDist := fSearchLineDist.Value,
    nMaxThickness := nMaxThickness.Value,
    nSubpixelsIterations := nSubpixelsIterations.Value,
    fApproxPrecision := fApproxPrecision.Value,
    eAlgorithm := eAlgorithm.Value,
    fRangeCutoffFactor := fRangeCutoffFactor.Value,
    ipEdgeStrengths := ipEdgeStrengths.Value,
    bAvgEdgeStrengths := bAvgEdgeStrengths.Value,
    hrPrev := hrPrev.Value,
    fAvgStrength => avgStrength);

fAvgStrength.Value := avgStrength;
END_METHOD

METHOD PUBLIC PreExecutionCheck
VAR_INPUT
    Check : I_PreExecutionChecks;
END_VAR
Check.IsTrue(ipSrcImage.IsValid, 'ipSrcImage must contain an image');
Check.IsTrue(ipSrcImage.HasChannelCount(1), 'ipSrcImage must contain 1 channel');
Check.IsTrue(nNumEdges.Value > 0, 'nNumEdges must be at least 1');
Check.IsTrue(nSearchLines.IsOdd, 'nSearchLines must be an odd number');
Check.IsTrue(fSearchLineDist.Value > 0.0, 'fSearchLineDist must be greater than 0');
Check.IsTrue(nMaxThickness.Value > 0, 'nMaxThickness must be at least 1');
Check.IsTrue(nSubpixelsIterations.Value > 0, 'nSubpixelsIterations must be greater than 0');
Check.IsTrue((eAlgorithm.Value = ETcVnEdgeDetectionAlgorithm.TCVN_EDA_INTERPOLATION) OR
             (fApproxPrecision.Value > 0.0), 'fApproxPrecision must be greater than 0 for the approximation algorithms');
END_METHOD

END_FUNCTION_BLOCK

// Nodes/Measurement/Node_F_VN_LocateEllipse
{attribute 'linkalways'} 
{attribute 'no_explicit_call' := 'This FB is a CLASS and must be accessed using methods or properties'}
{attribute 'enable_dynamic_creation'}
FUNCTION_BLOCK Node_F_VN_LocateEllipse EXTENDS VisionNode
VAR
	ipSrcImage : _ITcVnImage;
    stEllipse : _TcVnRotatedRectangle;
    aCenter : _TcVnPoint2_REAL;
    fSearchRadius : _REAL(0.0);
	eEdgeDirection : _ETcVnEdgeDirection(ETcVnEdgeDirection.TCVN_ED_DARK_TO_LIGHT);
    fMinStrength : _REAL(0.0);
    hrPrev : _HRESULT(S_OK);
	hresult : _HRESULT(S_OK);
END_VAR

METHOD FB_init : BOOL
VAR_INPUT
	bInitRetains : BOOL; // if TRUE, the retain variables are initialized (warm start / cold start)
	bInCopyCode : BOOL;  // if TRUE, the instance afterwards gets moved into the copy code (online change)
END_VAR
AddInput('ipSrcImage', ipSrcImage);
AddInput('aCenter', aCenter);
AddParameter('fSearchRadius', fSearchRadius);
AddParameter('eEdgeDirection', eEdgeDirection);
AddParameter('fMinStrength', fMinStrength);
AddInput('hrPrev', hrPrev);
AddOutput('stEllipse', stEllipse);
AddOutput('hresult',hresult);
END_METHOD

METHOD PUBLIC  Clone : I_Node
VAR
	pNode : POINTER TO Node_F_VN_LocateEllipse;
END_VAR
pNode := __NEW(Node_F_VN_LocateEllipse);
Clone := pNode^;
END_METHOD

METHOD PROTECTED OnExecute
hresult.Value := F_VN_LocateEllipse(
	ipSrcImage := ipSrcImage.Value,
    stEllipse := stEllipse.Value,
    aCenter := aCenter.Value,
    fSearchRadius := fSearchRadius.Value,
    eEdgeDirection := eEdgeDirection.Value,
	fMinStrength := fMinStrength.Value,
	hrPrev:= hrPrev.Value);
END_METHOD

METHOD PUBLIC PreExecutionCheck
VAR_INPUT
	Check : I_PreExecutionChecks;
END_VAR
Check.IsTrue(ipSrcImage.IsValid, 'ipSrcImage must contain an image');
Check.IsTrue(ipSrcImage.HasChannelCount(1), 'ipSrcImage must contain 1 channel');
END_METHOD

END_FUNCTION_BLOCK

// Nodes/Measurement/Node_F_VN_LocateEllipseExp
{attribute 'linkalways'} 
{attribute 'no_explicit_call' := 'This FB is a CLASS and must be accessed using methods or properties'}
{attribute 'enable_dynamic_creation'}
FUNCTION_BLOCK Node_F_VN_LocateEllipseExp EXTENDS VisionNode
VAR
	ipSrcImage : _ITcVnImage;
    stEllipse : _TcVnRotatedRectangle;
    aCenter : _TcVnPoint2_REAL;
    fSearchRadius : _REAL(0.0);
	eEdgeDirection : _ETcVnEdgeDirection(ETcVnEdgeDirection.TCVN_ED_DARK_TO_LIGHT);
    fMinStrength : _REAL(0.0);
	nMaxThickness : _UDINT(1);
	fMinSearchRadius : _REAL(0.0);
	bInvertSearchDirection : _BOOL(FALSE);
	nSubpixelsIterations : _UDINT(10);
	nSearchLines : _UDINT(1);
	fApproxPrecision : _REAL(0.001);
	eAlgorithm : _ETcVnEdgeDetectionAlgorithm(ETcVnEdgeDetectionAlgorithm.TCVN_EDA_APPROX_ERF);
	ipContourPoints : _ITcVnContainer;
    hrPrev : _HRESULT(S_OK);
	hresult : _HRESULT(S_OK);
END_VAR

METHOD FB_init : BOOL
VAR_INPUT
	bInitRetains : BOOL; // if TRUE, the retain variables are initialized (warm start / cold start)
	bInCopyCode : BOOL;  // if TRUE, the instance afterwards gets moved into the copy code (online change)
END_VAR
AddInput('ipSrcImage', ipSrcImage);
AddInput('aCenter', aCenter);
AddInput('hrPrev', hrPrev);
AddParameter('fSearchRadius', fSearchRadius);
AddParameter('eEdgeDirection', eEdgeDirection);
AddParameter('fMinStrength', fMinStrength);
AddParameter('nMaxThickness', nMaxThickness);
AddParameter('bInvertSearchDirection', bInvertSearchDirection);
AddParameter('fMinSearchRadius', fMinSearchRadius);
AddParameter('nSubpixelsIterations', nSubpixelsIterations);
AddParameter('nSearchLines', nSearchLines);
AddParameter('fApproxPrecision', fApproxPrecision);
AddParameter('eAlgorithm', eAlgorithm);
AddOutput('stEllipse', stEllipse);
AddOutput('aCenter', aCenter);
AddOutput('ipContourPoints', ipContourPoints);
AddOutput('hresult',hresult);
END_METHOD

METHOD PUBLIC  Clone : I_Node
VAR
	pNode : POINTER TO Node_F_VN_LocateEllipseExp;
END_VAR
pNode := __NEW(Node_F_VN_LocateEllipseExp);
Clone := pNode^;
END_METHOD

METHOD PROTECTED OnExecute
hresult.Value := F_VN_LocateEllipseExp(
	ipSrcImage := ipSrcImage.Value,
    stEllipse := stEllipse.Value,
    aCenter := aCenter.Value,
    fSearchRadius := fSearchRadius.Value,
    eEdgeDirection := eEdgeDirection.Value,
	fMinStrength := fMinStrength.Value,
	nMaxThickness := nMaxThickness.Value,
	bInvertSearchDirection := bInvertSearchDirection.Value,
	fMinSearchRadius := fMinSearchRadius.Value,
	nSubpixelsIterations := nSubpixelsIterations.Value,
	nSearchLines := nSearchLines.Value,
	fApproxPrecision := fApproxPrecision.Value,
	eAlgorithm := eAlgorithm.Value,
	ipContourPoints := ipContourPoints.Value,
	hrPrev:= hrPrev.Value);
END_METHOD

METHOD PUBLIC PreExecutionCheck
VAR_INPUT
	Check : I_PreExecutionChecks;
END_VAR
Check.IsTrue(ipSrcImage.IsValid, 'ipSrcImage must contain an image');
Check.IsTrue(ipSrcImage.HasChannelCount(1), 'ipSrcImage must contain 1 channel');

// Specifies the amount of search lines, which are equally distributed in all directions (must be >= 8 and a multiple of 4)
Check.IsTrue(nSearchLines.Value >= 8, 'nSearchLines must be >= 8');
Check.IsTrue(nSearchLines.Value MOD 4 = 0, 'nSearchLines must be a multiple of 4');
END_METHOD

END_FUNCTION_BLOCK

// Nodes/Measurement/Node_F_VN_LocateEllipseExp2
{attribute 'linkalways'}
{attribute 'no_explicit_call' := 'This FB is a CLASS and must be accessed using methods or properties'}
{attribute 'enable_dynamic_creation'}
FUNCTION_BLOCK Node_F_VN_LocateEllipseExp2 EXTENDS VisionNode
VAR
    ipSrcImage : _ITcVnImage;
    stEllipse : _TcVnRotatedRectangle;
    aCenter : _TcVnPoint2_REAL;
    fSearchRadius : _REAL(0.0);
    eEdgeDirection : _ETcVnEdgeDirection(ETcVnEdgeDirection.TCVN_ED_DARK_TO_LIGHT);
    fMinStrength : _REAL(0.0);
    nMaxThickness : _UDINT(10);
    bInvertSearchDirection : _BOOL(FALSE);
    fMinSearchRadius : _REAL(0.0);
    nSubpixelsIterations : _UDINT(10);
    nSearchLines : _UDINT(92);
    fApproxPrecision : _REAL(0.001);
    eAlgorithm : _ETcVnEdgeDetectionAlgorithm(ETcVnEdgeDetectionAlgorithm.TCVN_EDA_INTERPOLATION);
    ipContourPoints : _ITcVnContainer;
    fRangeCutoffFactor : _REAL(0.135);
    hrPrev : _HRESULT(S_OK);
    hresult : _HRESULT(S_OK);
END_VAR

METHOD FB_init : BOOL
VAR_INPUT
    bInitRetains : BOOL;
    bInCopyCode : BOOL;
END_VAR
AddInput('ipSrcImage', ipSrcImage);
AddOutput('stEllipse', stEllipse);
AddInput('aCenter', aCenter);
AddParameter('fSearchRadius', fSearchRadius);
AddParameter('eEdgeDirection', eEdgeDirection);
AddParameter('fMinStrength', fMinStrength);
AddParameter('nMaxThickness', nMaxThickness);
AddParameter('bInvertSearchDirection', bInvertSearchDirection);
AddParameter('fMinSearchRadius', fMinSearchRadius);
AddParameter('nSubpixelsIterations', nSubpixelsIterations);
AddParameter('nSearchLines', nSearchLines);
AddParameter('fApproxPrecision', fApproxPrecision);
AddParameter('eAlgorithm', eAlgorithm);
AddOutput('ipContourPoints', ipContourPoints);
AddParameter('fRangeCutoffFactor', fRangeCutoffFactor);
AddInput('hrPrev', hrPrev);
AddOutput('aCenter', aCenter);
AddOutput('hresult', hresult);
END_METHOD

METHOD PUBLIC Clone : I_Node
VAR
    pNode : POINTER TO Node_F_VN_LocateEllipseExp2;
END_VAR
pNode := __NEW(Node_F_VN_LocateEllipseExp2);
Clone := pNode^;
END_METHOD

METHOD PROTECTED OnExecute
hresult.Value := F_VN_LocateEllipseExp2(
    ipSrcImage := ipSrcImage.Value,
    stEllipse := stEllipse.Value,
    aCenter := aCenter.Value,
    fSearchRadius := fSearchRadius.Value,
    eEdgeDirection := eEdgeDirection.Value,
    fMinStrength := fMinStrength.Value,
    nMaxThickness := nMaxThickness.Value,
    bInvertSearchDirection := bInvertSearchDirection.Value,
    fMinSearchRadius := fMinSearchRadius.Value,
    nSubpixelsIterations := nSubpixelsIterations.Value,
    nSearchLines := nSearchLines.Value,
    fApproxPrecision := fApproxPrecision.Value,
    eAlgorithm := eAlgorithm.Value,
    ipContourPoints := ipContourPoints.Value,
    fRangeCutoffFactor := fRangeCutoffFactor.Value,
    hrPrev := hrPrev.Value);
END_METHOD

METHOD PUBLIC PreExecutionCheck
VAR_INPUT
    Check : I_PreExecutionChecks;
END_VAR
VAR
    width : UDINT;
    height : UDINT;
    cx : REAL;
    cy : REAL;
END_VAR
Check.IsTrue(ipSrcImage.IsValid, 'ipSrcImage must contain an image');
Check.IsTrue(ipSrcImage.HasChannelCount(1), 'ipSrcImage must contain 1 channel');

// Input search radius (starting FROM aCenter, should be greater than the actual radius but
// aCenter + fSearchRadius should be within the image borders)
ipSrcImage.TryGetWidth(width);
ipSrcImage.TryGetHeight(height);

Check.IsTrue((width > 0), 'ipSrcImage have valid width');
Check.IsTrue((height > 0), 'ipSrcImage have valid height');
Check.IsTrue(fSearchRadius.Value > 0, 'fSearchRadius must be > 0');

cx := aCenter.Value[0];
cy := aCenter.Value[1];

Check.IsTrue(cx - fSearchRadius.Value >= 0, 'Search radius exceeds left border');
Check.IsTrue(cy - fSearchRadius.Value >= 0, 'Search radius exceeds top border');
Check.IsTrue(cx + fSearchRadius.Value < UDINT_TO_REAL(width), 'Search radius exceeds right border');
Check.IsTrue(cy + fSearchRadius.Value < UDINT_TO_REAL(height), 'Search radius exceeds bottom border');

Check.IsTrue(nSearchLines.Value >= 8, 'nSearchLines must be >= 8');
Check.IsTrue(nSearchLines.Value MOD 4 = 0, 'nSearchLines must be a multiple of 4');
Check.IsTrue(fMinSearchRadius.Value >= 0.0, 'fMinSearchRadius cannot be negative');
Check.IsTrue(fMinSearchRadius.Value < fSearchRadius.Value, 'fMinSearchRadius must be smaller than fSearchRadius');

Check.IsTrue(nMaxThickness.Value > 0, 'nMaxThickness must be at least 1');
Check.IsTrue(nSubpixelsIterations.Value > 0, 'nSubpixelsIterations must be greater than 0');
Check.IsTrue((eAlgorithm.Value = ETcVnEdgeDetectionAlgorithm.TCVN_EDA_INTERPOLATION) OR
             (fApproxPrecision.Value > 0.0), 'fApproxPrecision must be greater than 0 for the approximation algorithms');
END_METHOD

END_FUNCTION_BLOCK

// Nodes/Measurement/Node_F_VN_MeasureAngleBetweenEdges
{attribute 'linkalways'} 
{attribute 'no_explicit_call' := 'This FB is a CLASS and must be accessed using methods or properties'}
{attribute 'enable_dynamic_creation'}
FUNCTION_BLOCK Node_F_VN_MeasureAngleBetweenEdges EXTENDS VisionNode
VAR
	ipSrcImage : _ITcVnImage;
    fAngle : _REAL(0.0);
    aInnerPoint : _TcVnPoint2_REAL;
    aOuterPoint1 : _TcVnPoint2_REAL;
    aOuterPoint2 : _TcVnPoint2_REAL;
	eEdgeDirection : _ETcVnEdgeDirection(ETcVnEdgeDirection.TCVN_ED_DARK_TO_LIGHT);
    fMinStrength : _REAL(0.0);
    nSearchLines : _UDINT(1);
    hrPrev : _HRESULT(S_OK);
	hresult : _HRESULT(S_OK);
END_VAR

METHOD FB_init : BOOL
VAR_INPUT
	bInitRetains : BOOL; // if TRUE, the retain variables are initialized (warm start / cold start)
	bInCopyCode : BOOL;  // if TRUE, the instance afterwards gets moved into the copy code (online change)
END_VAR
AddInput('ipSrcImage', ipSrcImage);
AddInput('aInnerPoint', aInnerPoint);
AddInput('aOuterPoint1', aOuterPoint1);
AddInput('aOuterPoint2', aOuterPoint2);
AddParameter('eEdgeDirection', eEdgeDirection);
AddParameter('fMinStrength', fMinStrength);
AddParameter('nSearchLines', nSearchLines);
AddInput('hrPrev', hrPrev);
AddOutput('fAngle', fAngle);
AddOutput('hresult',hresult);
END_METHOD

METHOD PUBLIC  Clone : I_Node
VAR
	pNode : POINTER TO Node_F_VN_MeasureAngleBetweenEdges;
END_VAR
pNode := __NEW(Node_F_VN_MeasureAngleBetweenEdges);
Clone := pNode^;
END_METHOD

METHOD PROTECTED OnExecute
hresult.Value := F_VN_MeasureAngleBetweenEdges(
	ipSrcImage := ipSrcImage.Value,
    fAngle := fAngle.Value,
	aInnerPoint := aInnerPoint.Value,
    aOuterPoint1 := aOuterPoint1.Value,
    aOuterPoint2 := aOuterPoint2.Value,
    eEdgeDirection := eEdgeDirection.Value,
	fMinStrength := fMinStrength.Value,
	nSearchLines := nSearchLines.Value,
	hrPrev:= hrPrev.Value);
END_METHOD

METHOD PUBLIC PreExecutionCheck
VAR_INPUT
	Check : I_PreExecutionChecks;
END_VAR
Check.IsTrue(ipSrcImage.IsValid, 'ipSrcImage must contain an image');
Check.IsTrue(ipSrcImage.HasChannelCount(1), 'ipSrcImage must contain 1 channel');
Check.IsTrue(nSearchLines.IsOdd, 'nSearchLines must be an odd number');
END_METHOD

END_FUNCTION_BLOCK

// Nodes/Measurement/Node_F_VN_MeasureAngleBetweenEdgesExp
{attribute 'linkalways'}
{attribute 'no_explicit_call' := 'This FB is a CLASS and must be accessed using methods or properties'}
{attribute 'enable_dynamic_creation'}
FUNCTION_BLOCK Node_F_VN_MeasureAngleBetweenEdgesExp EXTENDS VisionNode
VAR
    ipSrcImage : _ITcVnImage;
    fAngle : _REAL(0.0);
    aInnerPoint : _TcVnPoint2_REAL;
    aOuterPoint1 : _TcVnPoint2_REAL;
    aOuterPoint2 : _TcVnPoint2_REAL;
    eEdgeDirection : _ETcVnEdgeDirection(ETcVnEdgeDirection.TCVN_ED_DARK_TO_LIGHT);
    fMinStrength : _REAL(0.0);
    nSearchLines : _UDINT(3);
    fSearchLineDist : _REAL(1.0);
    nMaxThickness : _UDINT(10);
    bInvertSearchDirection : _BOOL(FALSE);
    nSubpixelsIterations : _UDINT(10);
    bAngleInDegrees : _BOOL(FALSE);
    fApproxPrecision : _REAL(0.001);
    eAlgorithm : _ETcVnEdgeDetectionAlgorithm(ETcVnEdgeDetectionAlgorithm.TCVN_EDA_INTERPOLATION);
    ipEdgePoints1 : _ITcVnContainer;
    ipEdgePoints2 : _ITcVnContainer;
    hrPrev : _HRESULT(S_OK);
    hresult : _HRESULT(S_OK);
END_VAR

METHOD FB_init : BOOL
VAR_INPUT
    bInitRetains : BOOL;
    bInCopyCode : BOOL;
END_VAR
AddInput('ipSrcImage', ipSrcImage);
AddOutput('fAngle', fAngle);
AddInput('aInnerPoint', aInnerPoint);
AddInput('aOuterPoint1', aOuterPoint1);
AddInput('aOuterPoint2', aOuterPoint2);
AddParameter('eEdgeDirection', eEdgeDirection);
AddParameter('fMinStrength', fMinStrength);
AddParameter('nSearchLines', nSearchLines);
AddParameter('fSearchLineDist', fSearchLineDist);
AddParameter('nMaxThickness', nMaxThickness);
AddParameter('bInvertSearchDirection', bInvertSearchDirection);
AddParameter('nSubpixelsIterations', nSubpixelsIterations);
AddParameter('bAngleInDegrees', bAngleInDegrees);
AddParameter('fApproxPrecision', fApproxPrecision);
AddParameter('eAlgorithm', eAlgorithm);
AddOutput('ipEdgePoints1', ipEdgePoints1);
AddOutput('ipEdgePoints2', ipEdgePoints2);
AddInput('hrPrev', hrPrev);
AddOutput('hresult', hresult);
END_METHOD

METHOD PUBLIC Clone : I_Node
VAR
    pNode : POINTER TO Node_F_VN_MeasureAngleBetweenEdgesExp;
END_VAR
pNode := __NEW(Node_F_VN_MeasureAngleBetweenEdgesExp);
Clone := pNode^;
END_METHOD

METHOD PROTECTED OnExecute
hresult.Value := F_VN_MeasureAngleBetweenEdgesExp(
    ipSrcImage := ipSrcImage.Value,
    fAngle := fAngle.Value,
    aInnerPoint := aInnerPoint.Value,
    aOuterPoint1 := aOuterPoint1.Value,
    aOuterPoint2 := aOuterPoint2.Value,
    eEdgeDirection := eEdgeDirection.Value,
    fMinStrength := fMinStrength.Value,
    nSearchLines := nSearchLines.Value,
    fSearchLineDist := fSearchLineDist.Value,
    nMaxThickness := nMaxThickness.Value,
    bInvertSearchDirection := bInvertSearchDirection.Value,
    nSubpixelsIterations := nSubpixelsIterations.Value,
    bAngleInDegrees := bAngleInDegrees.Value,
    fApproxPrecision := fApproxPrecision.Value,
    eAlgorithm := eAlgorithm.Value,
    ipEdgePoints1 := ipEdgePoints1.Value,
    ipEdgePoints2 := ipEdgePoints2.Value,
    hrPrev := hrPrev.Value);
END_METHOD

METHOD PUBLIC PreExecutionCheck
VAR_INPUT
    Check : I_PreExecutionChecks;
END_VAR
Check.IsTrue(ipSrcImage.IsValid, 'ipSrcImage must contain an image');
Check.IsTrue(ipSrcImage.HasChannelCount(1), 'ipSrcImage must contain 1 channel');
Check.IsTrue(nSearchLines.IsOdd, 'nSearchLines must be an odd number');
Check.IsTrue(fSearchLineDist.Value > 0.0, 'fSearchLineDist must be greater than 0');
Check.IsTrue(nSearchLines.Value >= 3, 'nSearchLines must be at least 3');
Check.IsTrue(nMaxThickness.Value > 0, 'nMaxThickness must be at least 1');
Check.IsTrue(nSubpixelsIterations.Value > 0, 'nSubpixelsIterations must be greater than 0');
Check.IsTrue((eAlgorithm.Value = ETcVnEdgeDetectionAlgorithm.TCVN_EDA_INTERPOLATION) OR
             (fApproxPrecision.Value > 0.0), 'fApproxPrecision must be greater than 0 for the approximation algorithms');
END_METHOD

END_FUNCTION_BLOCK

// Nodes/Measurement/Node_F_VN_MeasureAngleBetweenEdgesExp2
{attribute 'linkalways'}
{attribute 'no_explicit_call' := 'This FB is a CLASS and must be accessed using methods or properties'}
{attribute 'enable_dynamic_creation'}
FUNCTION_BLOCK Node_F_VN_MeasureAngleBetweenEdgesExp2 EXTENDS VisionNode
VAR
    ipSrcImage : _ITcVnImage;
    fAngle : _REAL(0.0);
    aInnerPoint : _TcVnPoint2_REAL;
    aOuterPoint1 : _TcVnPoint2_REAL;
    aOuterPoint2 : _TcVnPoint2_REAL;
    eEdgeDirection : _ETcVnEdgeDirection(ETcVnEdgeDirection.TCVN_ED_DARK_TO_LIGHT);
    fMinStrength : _REAL(0.0);
    nSearchLines : _UDINT(3);
    fSearchLineDist : _REAL(1.0);
    nMaxThickness : _UDINT(10);
    bInvertSearchDirection : _BOOL(FALSE);
    nSubpixelsIterations : _UDINT(10);
    bAngleInDegrees : _BOOL(FALSE);
    fApproxPrecision : _REAL(0.001);
    eAlgorithm : _ETcVnEdgeDetectionAlgorithm(ETcVnEdgeDetectionAlgorithm.TCVN_EDA_INTERPOLATION);
    ipEdgePoints1 : _ITcVnContainer;
    ipEdgePoints2 : _ITcVnContainer;
    fRangeCutoffFactor : _REAL(0.135);
    hrPrev : _HRESULT(S_OK);
    hresult : _HRESULT(S_OK);
END_VAR

METHOD FB_init : BOOL
VAR_INPUT
    bInitRetains : BOOL;
    bInCopyCode : BOOL;
END_VAR
AddInput('ipSrcImage', ipSrcImage);
AddOutput('fAngle', fAngle);
AddInput('aInnerPoint', aInnerPoint);
AddInput('aOuterPoint1', aOuterPoint1);
AddInput('aOuterPoint2', aOuterPoint2);
AddParameter('eEdgeDirection', eEdgeDirection);
AddParameter('fMinStrength', fMinStrength);
AddParameter('nSearchLines', nSearchLines);
AddParameter('fSearchLineDist', fSearchLineDist);
AddParameter('nMaxThickness', nMaxThickness);
AddParameter('bInvertSearchDirection', bInvertSearchDirection);
AddParameter('nSubpixelsIterations', nSubpixelsIterations);
AddParameter('bAngleInDegrees', bAngleInDegrees);
AddParameter('fApproxPrecision', fApproxPrecision);
AddParameter('eAlgorithm', eAlgorithm);
AddOutput('ipEdgePoints1', ipEdgePoints1);
AddOutput('ipEdgePoints2', ipEdgePoints2);
AddParameter('fRangeCutoffFactor', fRangeCutoffFactor);
AddInput('hrPrev', hrPrev);
AddOutput('hresult', hresult);
END_METHOD

METHOD PUBLIC Clone : I_Node
VAR
    pNode : POINTER TO Node_F_VN_MeasureAngleBetweenEdgesExp2;
END_VAR
pNode := __NEW(Node_F_VN_MeasureAngleBetweenEdgesExp2);
Clone := pNode^;
END_METHOD

METHOD PROTECTED OnExecute
hresult.Value := F_VN_MeasureAngleBetweenEdgesExp2(
    ipSrcImage := ipSrcImage.Value,
    fAngle := fAngle.Value,
    aInnerPoint := aInnerPoint.Value,
    aOuterPoint1 := aOuterPoint1.Value,
    aOuterPoint2 := aOuterPoint2.Value,
    eEdgeDirection := eEdgeDirection.Value,
    fMinStrength := fMinStrength.Value,
    nSearchLines := nSearchLines.Value,
    fSearchLineDist := fSearchLineDist.Value,
    nMaxThickness := nMaxThickness.Value,
    bInvertSearchDirection := bInvertSearchDirection.Value,
    nSubpixelsIterations := nSubpixelsIterations.Value,
    bAngleInDegrees := bAngleInDegrees.Value,
    fApproxPrecision := fApproxPrecision.Value,
    eAlgorithm := eAlgorithm.Value,
    ipEdgePoints1 := ipEdgePoints1.Value,
    ipEdgePoints2 := ipEdgePoints2.Value,
    fRangeCutoffFactor := fRangeCutoffFactor.Value,
    hrPrev := hrPrev.Value);
END_METHOD

METHOD PUBLIC PreExecutionCheck
VAR_INPUT
    Check : I_PreExecutionChecks;
END_VAR
Check.IsTrue(ipSrcImage.IsValid, 'ipSrcImage must contain an image');
Check.IsTrue(ipSrcImage.HasChannelCount(1), 'ipSrcImage must contain 1 channel');
Check.IsTrue(nSearchLines.IsOdd, 'nSearchLines must be an odd number');
Check.IsTrue(fSearchLineDist.Value > 0.0, 'fSearchLineDist must be greater than 0');
Check.IsTrue(nSearchLines.Value >= 3, 'nSearchLines must be at least 3');
Check.IsTrue(nMaxThickness.Value > 0, 'nMaxThickness must be at least 1');
Check.IsTrue(nSubpixelsIterations.Value > 0, 'nSubpixelsIterations must be greater than 0');
Check.IsTrue((eAlgorithm.Value = ETcVnEdgeDetectionAlgorithm.TCVN_EDA_INTERPOLATION) OR
             (fApproxPrecision.Value > 0.0), 'fApproxPrecision must be greater than 0 for the approximation algorithms');
END_METHOD

END_FUNCTION_BLOCK

// Nodes/Measurement/Node_F_VN_MeasureEdgeDistance
{attribute 'linkalways'} 
{attribute 'no_explicit_call' := 'This FB is a CLASS and must be accessed using methods or properties'}
{attribute 'enable_dynamic_creation'}
FUNCTION_BLOCK Node_F_VN_MeasureEdgeDistance EXTENDS VisionNode
VAR
	ipSrcImage : _ITcVnImage;
    fAvgDistance : _REAL(0.0);
    aStartPoint : _TcVnPoint2_REAL;
    aEndPoint : _TcVnPoint2_REAL;
	eEdgeDirection : _ETcVnEdgeDirection(ETcVnEdgeDirection.TCVN_ED_DARK_TO_LIGHT);
    fMinStrength : _REAL(0.0);
    nSearchLines : _UDINT(1);
    hrPrev : _HRESULT(S_OK);
	hresult : _HRESULT(S_OK);
END_VAR

METHOD FB_init : BOOL
VAR_INPUT
	bInitRetains : BOOL; // if TRUE, the retain variables are initialized (warm start / cold start)
	bInCopyCode : BOOL;  // if TRUE, the instance afterwards gets moved into the copy code (online change)
END_VAR
AddInput('ipSrcImage', ipSrcImage);
AddInput('aStartPoint', aStartPoint);
AddInput('aEndPoint', aEndPoint);
AddParameter('eEdgeDirection', eEdgeDirection);
AddParameter('fMinStrength', fMinStrength);
AddParameter('nSearchLines', nSearchLines);
AddInput('hrPrev', hrPrev);
AddOutput('fAvgDistance', fAvgDistance);
AddOutput('hresult',hresult);
END_METHOD

METHOD PUBLIC  Clone : I_Node
VAR
	pNode : POINTER TO Node_F_VN_MeasureEdgeDistance;
END_VAR
pNode := __NEW(Node_F_VN_MeasureEdgeDistance);
Clone := pNode^;
END_METHOD

METHOD PROTECTED OnExecute
hresult.Value := F_VN_MeasureEdgeDistance(
	ipSrcImage := ipSrcImage.Value,
    fAvgDistance := fAvgDistance.Value,
	aStartPoint := aStartPoint.Value,
    aEndPoint := aEndPoint.Value,
    eEdgeDirection := eEdgeDirection.Value,
	fMinStrength := fMinStrength.Value,
	nSearchLines := nSearchLines.Value,
	hrPrev:= hrPrev.Value);
END_METHOD

METHOD PUBLIC PreExecutionCheck
VAR_INPUT
	Check : I_PreExecutionChecks;
END_VAR
Check.IsTrue(ipSrcImage.IsValid, 'ipSrcImage must contain an image');
Check.IsTrue(ipSrcImage.HasChannelCount(1), 'ipSrcImage must contain 1 channel');
Check.IsTrue(nSearchLines.IsOdd, 'nSearchLines must be an odd number');
END_METHOD

END_FUNCTION_BLOCK

// Nodes/Measurement/Node_F_VN_MeasureEdgeDistanceExp
{attribute 'linkalways'} 
{attribute 'no_explicit_call' := 'This FB is a CLASS and must be accessed using methods or properties'}
{attribute 'enable_dynamic_creation'}
FUNCTION_BLOCK Node_F_VN_MeasureEdgeDistanceExp EXTENDS VisionNode
VAR
	ipSrcImage : _ITcVnImage;
    fAvgDistance : _REAL(0.0);
    aStartPoint : _TcVnPoint2_REAL;
    aEndPoint : _TcVnPoint2_REAL;
	eEdgeDirection : _ETcVnEdgeDirection(ETcVnEdgeDirection.TCVN_ED_DARK_TO_LIGHT);
    fMinStrength : _REAL(0.0);
    nSearchLines : _UDINT(1);
	fSearchLineDist : _REAL(1.0);
    nMaxThickness : _UDINT(1);
    bInvertSearchDirection : _BOOL(FALSE);
    fSearchGap : _REAL(0.0);
    nSubpixelsIterations : _UDINT(1);
    fApproxPrecision : _REAL(0.001);
    eAlgorithm: _ETcVnEdgeDetectionAlgorithm(ETcVnEdgeDetectionAlgorithm.TCVN_EDA_INTERPOLATION);
    ipEdgePoints1 : _ITcVnContainer;
    ipEdgePoints2 : _ITcVnContainer;
    ipDistances : _ITcVnContainer;
    hrPrev : _HRESULT(S_OK);
	hresult : _HRESULT(S_OK);
END_VAR

METHOD FB_init : BOOL
VAR_INPUT
	bInitRetains : BOOL; // if TRUE, the retain variables are initialized (warm start / cold start)
	bInCopyCode : BOOL;  // if TRUE, the instance afterwards gets moved into the copy code (online change)
END_VAR
AddInput('ipSrcImage', ipSrcImage);
AddInput('aStartPoint', aStartPoint);
AddInput('aEndPoint', aEndPoint);
AddParameter('eEdgeDirection', eEdgeDirection);
AddParameter('fMinStrength', fMinStrength);
AddParameter('nSearchLines', nSearchLines);
AddParameter('fSearchLineDist', fSearchLineDist);
AddParameter('nMaxThickness', nMaxThickness);
AddParameter('bInvertSearchDirection', bInvertSearchDirection);
AddParameter('fSearchGap', fSearchGap);
AddParameter('nSubpixelsIterations', nSubpixelsIterations);
AddParameter('fApproxPrecision', fApproxPrecision);
AddParameter('eAlgorithm', eAlgorithm);
AddInput('hrPrev', hrPrev);
AddOutput('fAvgDistance', fAvgDistance);
AddOutput('ipEdgePoints1', ipEdgePoints1);
AddOutput('ipEdgePoints2', ipEdgePoints2);
AddOutput('ipDistances', ipDistances);
AddOutput('hresult',hresult);
END_METHOD

METHOD PUBLIC  Clone : I_Node
VAR
	pNode : POINTER TO Node_F_VN_MeasureEdgeDistanceExp;
END_VAR
pNode := __NEW(Node_F_VN_MeasureEdgeDistanceExp);
Clone := pNode^;
END_METHOD

METHOD PROTECTED OnExecute
hresult.Value := F_VN_MeasureEdgeDistanceExp(
	ipSrcImage := ipSrcImage.Value,
    fAvgDistance := fAvgDistance.Value,
	aStartPoint := aStartPoint.Value,
    aEndPoint := aEndPoint.Value,
    eEdgeDirection := eEdgeDirection.Value,
	fMinStrength := fMinStrength.Value,
	nSearchLines := nSearchLines.Value,
	fSearchLineDist := fSearchLineDist.Value,
	nMaxThickness := nMaxThickness.Value,
	bInvertSearchDirection := bInvertSearchDirection.Value,
	fSearchGap := fSearchGap.Value,
	nSubpixelsIterations := nSubpixelsIterations.Value,
	fApproxPrecision := fApproxPrecision.Value,
	eAlgorithm := eAlgorithm.Value,
	ipEdgePoints1 := ipEdgePoints1.Value,
	ipEdgePoints2 := ipEdgePoints2.Value,
	ipDistances := ipDistances.Value,
	hrPrev:= hrPrev.Value
);
END_METHOD

METHOD PUBLIC PreExecutionCheck
VAR_INPUT
	Check : I_PreExecutionChecks;
END_VAR
Check.IsTrue(ipSrcImage.IsValid, 'ipSrcImage must contain an image');
Check.IsTrue(ipSrcImage.HasChannelCount(1), 'ipSrcImage must contain 1 channel');
Check.IsTrue(nSearchLines.IsOdd, 'nSearchLines must be an odd number');
Check.IsTrue(fSearchLineDist.Value > 0.0, 'fSearchLineDist must be greater than 0');
Check.IsTrue(nMaxThickness.Value > 0, 'nMaxThickness must be at least 1');
Check.IsTrue(fSearchGap.Value >= 0.0, 'fSearchGap cannot be negative');
Check.IsTrue(nSubpixelsIterations.Value > 0, 'nSubpixelsIterations must be greater than 0');
END_METHOD

END_FUNCTION_BLOCK

// Nodes/Measurement/Node_F_VN_MeasureEdgeDistanceExp2
{attribute 'linkalways'}
{attribute 'no_explicit_call' := 'This FB is a CLASS and must be accessed using methods or properties'}
{attribute 'enable_dynamic_creation'}
FUNCTION_BLOCK Node_F_VN_MeasureEdgeDistanceExp2 EXTENDS VisionNode
VAR
    ipSrcImage : _ITcVnImage;
    fAvgDistance : _REAL(0.0);
    aStartPoint : _TcVnPoint2_REAL;
    aEndPoint : _TcVnPoint2_REAL;
    eEdgeDirection : _ETcVnEdgeDirection(ETcVnEdgeDirection.TCVN_ED_DARK_TO_LIGHT);
    fMinStrength : _REAL(0.0);
    nSearchLines : _UDINT(1);
    fSearchLineDist : _REAL(1.0);
    nMaxThickness : _UDINT(10);
    bInvertSearchDirection : _BOOL(FALSE);
    fSearchGap : _REAL(0.0);
    nSubpixelsIterations : _UDINT(10);
    fApproxPrecision : _REAL(0.001);
    eAlgorithm : _ETcVnEdgeDetectionAlgorithm(ETcVnEdgeDetectionAlgorithm.TCVN_EDA_INTERPOLATION);
    ipEdgePoints1 : _ITcVnContainer;
    ipEdgePoints2 : _ITcVnContainer;
    ipDistances : _ITcVnContainer;
    fRangeCutoffFactor : _REAL(0.135);
    hrPrev : _HRESULT(S_OK);
    hresult : _HRESULT(S_OK);
END_VAR

METHOD FB_init : BOOL
VAR_INPUT
    bInitRetains : BOOL;
    bInCopyCode : BOOL;
END_VAR
AddInput('ipSrcImage', ipSrcImage);
AddOutput('fAvgDistance', fAvgDistance);
AddInput('aStartPoint', aStartPoint);
AddInput('aEndPoint', aEndPoint);
AddParameter('eEdgeDirection', eEdgeDirection);
AddParameter('fMinStrength', fMinStrength);
AddParameter('nSearchLines', nSearchLines);
AddParameter('fSearchLineDist', fSearchLineDist);
AddParameter('nMaxThickness', nMaxThickness);
AddParameter('bInvertSearchDirection', bInvertSearchDirection);
AddParameter('fSearchGap', fSearchGap);
AddParameter('nSubpixelsIterations', nSubpixelsIterations);
AddParameter('fApproxPrecision', fApproxPrecision);
AddParameter('eAlgorithm', eAlgorithm);
AddOutput('ipEdgePoints1', ipEdgePoints1);
AddOutput('ipEdgePoints2', ipEdgePoints2);
AddOutput('ipDistances', ipDistances);
AddParameter('fRangeCutoffFactor', fRangeCutoffFactor);
AddInput('hrPrev', hrPrev);
AddOutput('hresult', hresult);
END_METHOD

METHOD PUBLIC Clone : I_Node
VAR
    pNode : POINTER TO Node_F_VN_MeasureEdgeDistanceExp2;
END_VAR
pNode := __NEW(Node_F_VN_MeasureEdgeDistanceExp2);
Clone := pNode^;
END_METHOD

METHOD PROTECTED OnExecute
hresult.Value := F_VN_MeasureEdgeDistanceExp2(
    ipSrcImage := ipSrcImage.Value,
    fAvgDistance := fAvgDistance.Value,
    aStartPoint := aStartPoint.Value,
    aEndPoint := aEndPoint.Value,
    eEdgeDirection := eEdgeDirection.Value,
    fMinStrength := fMinStrength.Value,
    nSearchLines := nSearchLines.Value,
    fSearchLineDist := fSearchLineDist.Value,
    nMaxThickness := nMaxThickness.Value,
    bInvertSearchDirection := bInvertSearchDirection.Value,
    fSearchGap := fSearchGap.Value,
    nSubpixelsIterations := nSubpixelsIterations.Value,
    fApproxPrecision := fApproxPrecision.Value,
    eAlgorithm := eAlgorithm.Value,
    ipEdgePoints1 := ipEdgePoints1.Value,
    ipEdgePoints2 := ipEdgePoints2.Value,
    ipDistances := ipDistances.Value,
    fRangeCutoffFactor := fRangeCutoffFactor.Value,
    hrPrev := hrPrev.Value);
END_METHOD

METHOD PUBLIC PreExecutionCheck
VAR_INPUT
    Check : I_PreExecutionChecks;
END_VAR
Check.IsTrue(ipSrcImage.IsValid, 'ipSrcImage must contain an image');
Check.IsTrue(ipSrcImage.HasChannelCount(1), 'ipSrcImage must contain 1 channel');
Check.IsTrue(nSearchLines.IsOdd, 'nSearchLines must be an odd number');
Check.IsTrue(fSearchLineDist.Value > 0.0, 'fSearchLineDist must be greater than 0');
Check.IsTrue(fSearchGap.Value >= 0.0, 'fSearchGap cannot be negative');
Check.IsTrue(nMaxThickness.Value > 0, 'nMaxThickness must be at least 1');
Check.IsTrue(nSubpixelsIterations.Value > 0, 'nSubpixelsIterations must be greater than 0');
Check.IsTrue((eAlgorithm.Value = ETcVnEdgeDetectionAlgorithm.TCVN_EDA_INTERPOLATION) OR
             (fApproxPrecision.Value > 0.0), 'fApproxPrecision must be greater than 0 for the approximation algorithms');
END_METHOD

END_FUNCTION_BLOCK

// Nodes/Measurement/Node_F_VN_MeasureMinEdgeDistance
{attribute 'linkalways'} 
{attribute 'no_explicit_call' := 'This FB is a CLASS and must be accessed using methods or properties'}
{attribute 'enable_dynamic_creation'}
FUNCTION_BLOCK Node_F_VN_MeasureMinEdgeDistance EXTENDS VisionNode
VAR
	ipSrcImage : _ITcVnImage;
    fMinDistance : _REAL(0.0);
    aStartPoint : _TcVnPoint2_REAL;
    aEndPoint : _TcVnPoint2_REAL;
	eEdgeDirection : _ETcVnEdgeDirection(ETcVnEdgeDirection.TCVN_ED_DARK_TO_LIGHT);
    fMinStrength : _REAL(0.0);
    nSearchLines : _UDINT(1);
    hrPrev : _HRESULT(S_OK);
	hresult : _HRESULT(S_OK);
END_VAR

METHOD FB_init : BOOL
VAR_INPUT
	bInitRetains : BOOL; // if TRUE, the retain variables are initialized (warm start / cold start)
	bInCopyCode : BOOL;  // if TRUE, the instance afterwards gets moved into the copy code (online change)
END_VAR
AddInput('ipSrcImage', ipSrcImage);
AddInput('aStartPoint', aStartPoint);
AddInput('aEndPoint', aEndPoint);
AddParameter('eEdgeDirection', eEdgeDirection);
AddParameter('fMinStrength', fMinStrength);
AddParameter('nSearchLines', nSearchLines);
AddInput('hrPrev', hrPrev);
AddOutput('fMinDistance', fMinDistance);
AddOutput('hresult',hresult);
END_METHOD

METHOD PUBLIC  Clone : I_Node
VAR
	pNode : POINTER TO Node_F_VN_MeasureMinEdgeDistance;
END_VAR
pNode := __NEW(Node_F_VN_MeasureMinEdgeDistance);
Clone := pNode^;
END_METHOD

METHOD PROTECTED OnExecute
hresult.Value := F_VN_MeasureMinEdgeDistance(
	ipSrcImage := ipSrcImage.Value,
    fMinDistance := fMinDistance.Value,
	aStartPoint := aStartPoint.Value,
    aEndPoint := aEndPoint.Value,
    eEdgeDirection := eEdgeDirection.Value,
	fMinStrength := fMinStrength.Value,
	nSearchLines := nSearchLines.Value,
	hrPrev:= hrPrev.Value);
END_METHOD

METHOD PUBLIC PreExecutionCheck
VAR_INPUT
	Check : I_PreExecutionChecks;
END_VAR
Check.IsTrue(ipSrcImage.IsValid, 'ipSrcImage must contain an image');
Check.IsTrue(ipSrcImage.HasChannelCount(1), 'ipSrcImage must contain 1 channel');
Check.IsTrue(nSearchLines.IsOdd, 'nSearchLines must be an odd number');
END_METHOD

END_FUNCTION_BLOCK

// Nodes/Measurement/Node_F_VN_MeasureMinEdgeDistanceExp
{attribute 'linkalways'}
{attribute 'no_explicit_call' := 'This FB is a CLASS and must be accessed using methods or properties'}
{attribute 'enable_dynamic_creation'}
FUNCTION_BLOCK Node_F_VN_MeasureMinEdgeDistanceExp EXTENDS VisionNode
VAR
    ipSrcImage : _ITcVnImage;
    fMinDistance : _REAL(0.0);
    aStartPoint : _TcVnPoint2_REAL;
    aEndPoint : _TcVnPoint2_REAL;
    eEdgeDirection : _ETcVnEdgeDirection(ETcVnEdgeDirection.TCVN_ED_DARK_TO_LIGHT);
    fMinStrength : _REAL(0.0);
    nSearchLines : _UDINT(1);
    fSearchLineDist : _REAL(1.0);
    nMaxThickness : _UDINT(10);
    bInvertSearchDirection : _BOOL(FALSE);
    fSearchGap : _REAL(0.0);
    nSubpixelsIterations : _UDINT(10);
    fApproxPrecision : _REAL(0.001);
    eAlgorithm : _ETcVnEdgeDetectionAlgorithm(ETcVnEdgeDetectionAlgorithm.TCVN_EDA_INTERPOLATION);
    ipEdgePoints1 : _ITcVnContainer;
    ipEdgePoints2 : _ITcVnContainer;
    aPoint1 : _TcVnPoint2_REAL;
    aPoint2 : _TcVnPoint2_REAL;
    hrPrev : _HRESULT(S_OK);
    hresult : _HRESULT(S_OK);
END_VAR

METHOD FB_init : BOOL
VAR_INPUT
    bInitRetains : BOOL;
    bInCopyCode : BOOL;
END_VAR
AddInput('ipSrcImage', ipSrcImage);
AddOutput('fMinDistance', fMinDistance);
AddInput('aStartPoint', aStartPoint);
AddInput('aEndPoint', aEndPoint);
AddParameter('eEdgeDirection', eEdgeDirection);
AddParameter('fMinStrength', fMinStrength);
AddParameter('nSearchLines', nSearchLines);
AddParameter('fSearchLineDist', fSearchLineDist);
AddParameter('nMaxThickness', nMaxThickness);
AddParameter('bInvertSearchDirection', bInvertSearchDirection);
AddParameter('fSearchGap', fSearchGap);
AddParameter('nSubpixelsIterations', nSubpixelsIterations);
AddParameter('fApproxPrecision', fApproxPrecision);
AddParameter('eAlgorithm', eAlgorithm);
AddOutput('ipEdgePoints1', ipEdgePoints1);
AddOutput('ipEdgePoints2', ipEdgePoints2);
AddOutput('aPoint1', aPoint1);
AddOutput('aPoint2', aPoint2);
AddInput('hrPrev', hrPrev);
AddOutput('hresult', hresult);
END_METHOD

METHOD PUBLIC Clone : I_Node
VAR
    pNode : POINTER TO Node_F_VN_MeasureMinEdgeDistanceExp;
END_VAR
pNode := __NEW(Node_F_VN_MeasureMinEdgeDistanceExp);
Clone := pNode^;
END_METHOD

METHOD PROTECTED OnExecute
hresult.Value := F_VN_MeasureMinEdgeDistanceExp(
    ipSrcImage := ipSrcImage.Value,
    fMinDistance := fMinDistance.Value,
    aStartPoint := aStartPoint.Value,
    aEndPoint := aEndPoint.Value,
    eEdgeDirection := eEdgeDirection.Value,
    fMinStrength := fMinStrength.Value,
    nSearchLines := nSearchLines.Value,
    fSearchLineDist := fSearchLineDist.Value,
    nMaxThickness := nMaxThickness.Value,
    bInvertSearchDirection := bInvertSearchDirection.Value,
    fSearchGap := fSearchGap.Value,
    nSubpixelsIterations := nSubpixelsIterations.Value,
    fApproxPrecision := fApproxPrecision.Value,
    eAlgorithm := eAlgorithm.Value,
    ipEdgePoints1 := ipEdgePoints1.Value,
    ipEdgePoints2 := ipEdgePoints2.Value,
    aPoint1 := aPoint1.Value,
    aPoint2 := aPoint2.Value,
    hrPrev := hrPrev.Value);
END_METHOD

METHOD PUBLIC PreExecutionCheck
VAR_INPUT
    Check : I_PreExecutionChecks;
END_VAR
Check.IsTrue(ipSrcImage.IsValid, 'ipSrcImage must contain an image');
Check.IsTrue(ipSrcImage.HasChannelCount(1), 'ipSrcImage must contain 1 channel');
Check.IsTrue(nSearchLines.IsOdd, 'nSearchLines must be an odd number');
Check.IsTrue(fSearchLineDist.Value > 0.0, 'fSearchLineDist must be greater than 0');
Check.IsTrue(fSearchGap.Value >= 0.0, 'fSearchGap cannot be negative');
Check.IsTrue(nMaxThickness.Value > 0, 'nMaxThickness must be at least 1');
Check.IsTrue(nSubpixelsIterations.Value > 0, 'nSubpixelsIterations must be greater than 0');
Check.IsTrue((eAlgorithm.Value = ETcVnEdgeDetectionAlgorithm.TCVN_EDA_INTERPOLATION) OR
             (fApproxPrecision.Value > 0.0), 'fApproxPrecision must be greater than 0 for the approximation algorithms');
END_METHOD

END_FUNCTION_BLOCK

// Nodes/Measurement/Node_F_VN_MeasureMinEdgeDistanceExp2
{attribute 'linkalways'}
{attribute 'no_explicit_call' := 'This FB is a CLASS and must be accessed using methods or properties'}
{attribute 'enable_dynamic_creation'}
FUNCTION_BLOCK Node_F_VN_MeasureMinEdgeDistanceExp2 EXTENDS VisionNode
VAR
    ipSrcImage : _ITcVnImage;
    fMinDistance : _REAL(0.0);
    aStartPoint : _TcVnPoint2_REAL;
    aEndPoint : _TcVnPoint2_REAL;
    eEdgeDirection : _ETcVnEdgeDirection(ETcVnEdgeDirection.TCVN_ED_DARK_TO_LIGHT);
    fMinStrength : _REAL(0.0);
    nSearchLines : _UDINT(1);
    fSearchLineDist : _REAL(1.0);
    nMaxThickness : _UDINT(10);
    bInvertSearchDirection : _BOOL(FALSE);
    fSearchGap : _REAL(0.0);
    nSubpixelsIterations : _UDINT(10);
    fApproxPrecision : _REAL(0.001);
    eAlgorithm : _ETcVnEdgeDetectionAlgorithm(ETcVnEdgeDetectionAlgorithm.TCVN_EDA_INTERPOLATION);
    ipEdgePoints1 : _ITcVnContainer;
    ipEdgePoints2 : _ITcVnContainer;
    aPoint1 : _TcVnPoint2_REAL;
    aPoint2 : _TcVnPoint2_REAL;
    fRangeCutoffFactor : _REAL(0.135);
    hrPrev : _HRESULT(S_OK);
    hresult : _HRESULT(S_OK);
END_VAR

METHOD FB_init : BOOL
VAR_INPUT
    bInitRetains : BOOL;
    bInCopyCode : BOOL;
END_VAR
AddInput('ipSrcImage', ipSrcImage);
AddOutput('fMinDistance', fMinDistance);
AddInput('aStartPoint', aStartPoint);
AddInput('aEndPoint', aEndPoint);
AddParameter('eEdgeDirection', eEdgeDirection);
AddParameter('fMinStrength', fMinStrength);
AddParameter('nSearchLines', nSearchLines);
AddParameter('fSearchLineDist', fSearchLineDist);
AddParameter('nMaxThickness', nMaxThickness);
AddParameter('bInvertSearchDirection', bInvertSearchDirection);
AddParameter('fSearchGap', fSearchGap);
AddParameter('nSubpixelsIterations', nSubpixelsIterations);
AddParameter('fApproxPrecision', fApproxPrecision);
AddParameter('eAlgorithm', eAlgorithm);
AddOutput('ipEdgePoints1', ipEdgePoints1);
AddOutput('ipEdgePoints2', ipEdgePoints2);
AddOutput('aPoint1', aPoint1);
AddOutput('aPoint2', aPoint2);
AddParameter('fRangeCutoffFactor', fRangeCutoffFactor);
AddInput('hrPrev', hrPrev);
AddOutput('hresult', hresult);
END_METHOD

METHOD PUBLIC Clone : I_Node
VAR
    pNode : POINTER TO Node_F_VN_MeasureMinEdgeDistanceExp2;
END_VAR
pNode := __NEW(Node_F_VN_MeasureMinEdgeDistanceExp2);
Clone := pNode^;
END_METHOD

METHOD PROTECTED OnExecute
hresult.Value := F_VN_MeasureMinEdgeDistanceExp2(
    ipSrcImage := ipSrcImage.Value,
    fMinDistance := fMinDistance.Value,
    aStartPoint := aStartPoint.Value,
    aEndPoint := aEndPoint.Value,
    eEdgeDirection := eEdgeDirection.Value,
    fMinStrength := fMinStrength.Value,
    nSearchLines := nSearchLines.Value,
    fSearchLineDist := fSearchLineDist.Value,
    nMaxThickness := nMaxThickness.Value,
    bInvertSearchDirection := bInvertSearchDirection.Value,
    fSearchGap := fSearchGap.Value,
    nSubpixelsIterations := nSubpixelsIterations.Value,
    fApproxPrecision := fApproxPrecision.Value,
    eAlgorithm := eAlgorithm.Value,
    ipEdgePoints1 := ipEdgePoints1.Value,
    ipEdgePoints2 := ipEdgePoints2.Value,
    aPoint1 := aPoint1.Value,
    aPoint2 := aPoint2.Value,
    fRangeCutoffFactor := fRangeCutoffFactor.Value,
    hrPrev := hrPrev.Value);
END_METHOD

METHOD PUBLIC PreExecutionCheck
VAR_INPUT
    Check : I_PreExecutionChecks;
END_VAR
Check.IsTrue(ipSrcImage.IsValid, 'ipSrcImage must contain an image');
Check.IsTrue(ipSrcImage.HasChannelCount(1), 'ipSrcImage must contain 1 channel');
Check.IsTrue(nSearchLines.IsOdd, 'nSearchLines must be an odd number');
Check.IsTrue(fSearchLineDist.Value > 0.0, 'fSearchLineDist must be greater than 0');
Check.IsTrue(fSearchGap.Value >= 0.0, 'fSearchGap cannot be negative');
Check.IsTrue(nMaxThickness.Value > 0, 'nMaxThickness must be at least 1');
Check.IsTrue(nSubpixelsIterations.Value > 0, 'nSubpixelsIterations must be greater than 0');
Check.IsTrue((eAlgorithm.Value = ETcVnEdgeDetectionAlgorithm.TCVN_EDA_INTERPOLATION) OR
             (fApproxPrecision.Value > 0.0), 'fApproxPrecision must be greater than 0 for the approximation algorithms');
END_METHOD

END_FUNCTION_BLOCK

// Nodes/Miscellaneous/Node_F_VN_CheckFunctionInitialization
{attribute 'linkalways'} 
{attribute 'no_explicit_call' := 'This FB is a CLASS and must be accessed using methods or properties'}
{attribute 'enable_dynamic_creation'}
FUNCTION_BLOCK Node_F_VN_CheckFunctionInitialization EXTENDS VisionNode
VAR
    eFunction : _ETcVnInitializableFunction(ETcVnInitializableFunction.TCVN_IF_OCR);
    nOptions : _ULINT(0);
    hrPrev : _HRESULT(S_OK);
	hresult : _HRESULT(S_OK);
END_VAR

METHOD FB_init : BOOL
VAR_INPUT
	bInitRetains : BOOL; // if TRUE, the retain variables are initialized (warm start / cold start)
	bInCopyCode : BOOL;  // if TRUE, the instance afterwards gets moved into the copy code (online change)
END_VAR
AddParameter('eFunction', eFunction);
AddInput('nOptions', nOptions);
AddInput('hrPrev', hrPrev);
AddOutput('hresult',hresult);
END_METHOD

METHOD PUBLIC  Clone : I_Node
VAR
	pNode : POINTER TO Node_F_VN_CheckFunctionInitialization;
END_VAR
pNode := __NEW(Node_F_VN_CheckFunctionInitialization);
Clone := pNode^;
END_METHOD

METHOD PROTECTED OnExecute
hresult.Value := F_VN_CheckFunctionInitialization(
	eFunction := eFunction.Value,
    nOptions := nOptions.Value,
	hrPrev:= hrPrev.Value);
END_METHOD

METHOD PUBLIC PreExecutionCheck
VAR_INPUT
	Check : I_PreExecutionChecks;
END_VAR
END_METHOD

END_FUNCTION_BLOCK

// Nodes/Miscellaneous/Node_F_VN_ClipLineToBoundary
{attribute 'linkalways'} 
{attribute 'no_explicit_call' := 'This FB is a CLASS and must be accessed using methods or properties'}
{attribute 'enable_dynamic_creation'}
FUNCTION_BLOCK Node_F_VN_ClipLineToBoundary EXTENDS VisionNode
VAR
    aLine : _TcVnVector4_LREAL;
    nX1 : _DINT(0);
    nY1 : _DINT(0);
    nX2 : _DINT(0);
    nY2 : _DINT(0);
    aStartPoint : _TcVnPoint2_REAL;
    aEndPoint : _TcVnPoint2_REAL;
    hrPrev : _HRESULT(S_OK);
	hresult : _HRESULT(S_OK);
END_VAR

METHOD FB_init : BOOL
VAR_INPUT
	bInitRetains : BOOL; // if TRUE, the retain variables are initialized (warm start / cold start)
	bInCopyCode : BOOL;  // if TRUE, the instance afterwards gets moved into the copy code (online change)
END_VAR
AddInput('aLine', aLine);
AddParameter('nX1', nX1);
AddParameter('nY1', nY1);
AddParameter('nX2', nX2);
AddParameter('nY2', nY2);
AddInput('aStartPoint', aStartPoint);
AddInput('aEndPoint', aEndPoint);
AddInput('hrPrev', hrPrev);
AddOutput('aLine', aLine);
AddOutput('aStartPoint', aStartPoint);
AddOutput('aEndPoint', aEndPoint);
AddOutput('hresult',hresult);
END_METHOD

METHOD PUBLIC  Clone : I_Node
VAR
	pNode : POINTER TO Node_F_VN_ClipLineToBoundary;
END_VAR
pNode := __NEW(Node_F_VN_ClipLineToBoundary);
Clone := pNode^;
END_METHOD

METHOD PROTECTED OnExecute
hresult.Value := F_VN_ClipLineToBoundary(
	aLine := aLine.Value,
    nX1 := nX1.Value,
    nY1 := nY1.Value,
    nX2 := nX2.Value,
    nY2 := nY2.Value,
    aStartPoint := aStartPoint.Value,
    aEndPoint := aEndPoint.Value,
	hrPrev:= hrPrev.Value);
END_METHOD

METHOD PUBLIC PreExecutionCheck
VAR_INPUT
	Check : I_PreExecutionChecks;
END_VAR
END_METHOD

END_FUNCTION_BLOCK

// Nodes/Miscellaneous/Node_F_VN_ClipLineToBoundary_ITcVnImage
{attribute 'linkalways'} 
{attribute 'no_explicit_call' := 'This FB is a CLASS and must be accessed using methods or properties'}
{attribute 'enable_dynamic_creation'}
FUNCTION_BLOCK Node_F_VN_ClipLineToBoundary_ITcVnImage EXTENDS VisionNode
VAR
    aLine : _TcVnVector4_LREAL;
    ipImage : _ITcVnImage;
    aStartPoint : _TcVnPoint2_REAL;
    aEndPoint : _TcVnPoint2_REAL;
    hrPrev : _HRESULT(S_OK);
	hresult : _HRESULT(S_OK);
END_VAR

METHOD FB_init : BOOL
VAR_INPUT
	bInitRetains : BOOL; // if TRUE, the retain variables are initialized (warm start / cold start)
	bInCopyCode : BOOL;  // if TRUE, the instance afterwards gets moved into the copy code (online change)
END_VAR
AddInput('aLine', aLine);
AddInput('ipImage', ipImage);
AddInput('aStartPoint', aStartPoint);
AddInput('aEndPoint', aEndPoint);
AddInput('hrPrev', hrPrev);
AddOutput('aLine', aLine);
AddOutput('aStartPoint', aStartPoint);
AddOutput('aEndPoint', aEndPoint);
AddOutput('hresult',hresult);
END_METHOD

METHOD PUBLIC  Clone : I_Node
VAR
	pNode : POINTER TO Node_F_VN_ClipLineToBoundary_ITcVnImage;
END_VAR
pNode := __NEW(Node_F_VN_ClipLineToBoundary_ITcVnImage);
Clone := pNode^;
END_METHOD

METHOD PROTECTED OnExecute
hresult.Value := F_VN_ClipLineToBoundary_ITcVnImage(
	aLine := aLine.Value,
    ipImage := ipImage.Value,
    aStartPoint := aStartPoint.Value,
    aEndPoint := aEndPoint.Value,
	hrPrev:= hrPrev.Value);
END_METHOD

METHOD PUBLIC PreExecutionCheck
VAR_INPUT
	Check : I_PreExecutionChecks;
END_VAR
Check.IsTrue(ipImage.IsValid, 'ipImage must contain an image');
END_METHOD

END_FUNCTION_BLOCK

// Nodes/Miscellaneous/Node_F_VN_ClipLineToBoundary_TcVnRectangle_DINT
{attribute 'linkalways'} 
{attribute 'no_explicit_call' := 'This FB is a CLASS and must be accessed using methods or properties'}
{attribute 'enable_dynamic_creation'}
FUNCTION_BLOCK Node_F_VN_ClipLineToBoundary_TcVnRectangle_DINT EXTENDS VisionNode
VAR
    aLine : _TcVnVector4_LREAL;
    stRectangle : _TcVnRectangle_DINT;
    aStartPoint : _TcVnPoint2_REAL;
    aEndPoint : _TcVnPoint2_REAL;
    hrPrev : _HRESULT(S_OK);
	hresult : _HRESULT(S_OK);
END_VAR

METHOD FB_init : BOOL
VAR_INPUT
	bInitRetains : BOOL; // if TRUE, the retain variables are initialized (warm start / cold start)
	bInCopyCode : BOOL;  // if TRUE, the instance afterwards gets moved into the copy code (online change)
END_VAR
AddInput('aLine', aLine);
AddInput('stRectangle', stRectangle);
AddInput('aStartPoint', aStartPoint);
AddInput('aEndPoint', aEndPoint);
AddInput('hrPrev', hrPrev);
AddOutput('aLine', aLine);
AddOutput('aStartPoint', aStartPoint);
AddOutput('aEndPoint', aEndPoint);
AddOutput('hresult',hresult);
END_METHOD

METHOD PUBLIC  Clone : I_Node
VAR
	pNode : POINTER TO Node_F_VN_ClipLineToBoundary_TcVnRectangle_DINT;
END_VAR
pNode := __NEW(Node_F_VN_ClipLineToBoundary_TcVnRectangle_DINT);
Clone := pNode^;
END_METHOD

METHOD PROTECTED OnExecute
hresult.Value := F_VN_ClipLineToBoundary_TcVnRectangle_DINT(
	aLine := aLine.Value,
    stRectangle := stRectangle.Value,
    aStartPoint := aStartPoint.Value,
    aEndPoint := aEndPoint.Value,
	hrPrev:= hrPrev.Value);
END_METHOD

METHOD PUBLIC PreExecutionCheck
VAR_INPUT
	Check : I_PreExecutionChecks;
END_VAR
END_METHOD

END_FUNCTION_BLOCK

// Nodes/Miscellaneous/Node_F_VN_DeinitializeFunction
{attribute 'linkalways'} 
{attribute 'no_explicit_call' := 'This FB is a CLASS and must be accessed using methods or properties'}
{attribute 'enable_dynamic_creation'}
FUNCTION_BLOCK Node_F_VN_DeinitializeFunction EXTENDS VisionNode
VAR
    eFunction : _ETcVnInitializableFunction(ETcVnInitializableFunction.TCVN_IF_OCR);
    nOptions : _ULINT(0);
    hrPrev : _HRESULT(S_OK);
	hresult : _HRESULT(S_OK);
END_VAR

METHOD FB_init : BOOL
VAR_INPUT
	bInitRetains : BOOL; // if TRUE, the retain variables are initialized (warm start / cold start)
	bInCopyCode : BOOL;  // if TRUE, the instance afterwards gets moved into the copy code (online change)
END_VAR
AddParameter('eFunction', eFunction);
AddParameter('nOptions', nOptions);
AddInput('hrPrev', hrPrev);
AddOutput('hresult',hresult);
END_METHOD

METHOD PUBLIC  Clone : I_Node
VAR
	pNode : POINTER TO Node_F_VN_DeinitializeFunction;
END_VAR
pNode := __NEW(Node_F_VN_DeinitializeFunction);
Clone := pNode^;
END_METHOD

METHOD PROTECTED OnExecute
hresult.Value := F_VN_DeinitializeFunction(
	eFunction := eFunction.Value,
    nOptions := nOptions.Value,
	hrPrev:= hrPrev.Value);
END_METHOD

METHOD PUBLIC PreExecutionCheck
VAR_INPUT
	Check : I_PreExecutionChecks;
END_VAR
END_METHOD

END_FUNCTION_BLOCK

// Nodes/Miscellaneous/Node_F_VN_HuMomentInvariants
{attribute 'linkalways'} 
{attribute 'no_explicit_call' := 'This FB is a CLASS and must be accessed using methods or properties'}
{attribute 'enable_dynamic_creation'}
FUNCTION_BLOCK Node_F_VN_HuMomentInvariants EXTENDS VisionNode
VAR
    stMoments : _TcVnMoments;
    aHuInvariants : _TcVnArray7_LREAL;
    hrPrev : _HRESULT(S_OK);
	hresult : _HRESULT(S_OK);
END_VAR

METHOD FB_init : BOOL
VAR_INPUT
	bInitRetains : BOOL; // if TRUE, the retain variables are initialized (warm start / cold start)
	bInCopyCode : BOOL;  // if TRUE, the instance afterwards gets moved into the copy code (online change)
END_VAR
AddInput('stMoments', stMoments);
AddInput('hrPrev', hrPrev);
AddOutput('aHuInvariants', aHuInvariants);
AddOutput('hresult',hresult);
END_METHOD

METHOD PUBLIC  Clone : I_Node
VAR
	pNode : POINTER TO Node_F_VN_HuMomentInvariants;
END_VAR
pNode := __NEW(Node_F_VN_HuMomentInvariants);
Clone := pNode^;
END_METHOD

METHOD PROTECTED OnExecute
hresult.Value := F_VN_HuMomentInvariants(
	stMoments := stMoments.Value,
    aHuInvariants := aHuInvariants.Value,
	hrPrev:= hrPrev.Value);
END_METHOD

METHOD PUBLIC PreExecutionCheck
VAR_INPUT
	Check : I_PreExecutionChecks;
END_VAR
END_METHOD

END_FUNCTION_BLOCK

// Nodes/Miscellaneous/Node_F_VN_InvertMatrix3x3
{attribute 'linkalways'} 
{attribute 'no_explicit_call' := 'This FB is a CLASS and must be accessed using methods or properties'}
{attribute 'enable_dynamic_creation'}
FUNCTION_BLOCK Node_F_VN_InvertMatrix3x3 EXTENDS VisionNode
VAR
    aSrcMatrix : _TcVnMatrix3x3_LREAL;
    aInvertedMatrix : _TcVnMatrix3x3_LREAL;
    hrPrev : _HRESULT(S_OK);
	hresult : _HRESULT(S_OK);
END_VAR

METHOD FB_init : BOOL
VAR_INPUT
	bInitRetains : BOOL; // if TRUE, the retain variables are initialized (warm start / cold start)
	bInCopyCode : BOOL;  // if TRUE, the instance afterwards gets moved into the copy code (online change)
END_VAR
AddInput('aSrcMatrix', aSrcMatrix);
AddInput('hrPrev', hrPrev);
AddOutput('aInvertedMatrix', aInvertedMatrix);
AddOutput('hresult',hresult);
END_METHOD

METHOD PUBLIC  Clone : I_Node
VAR
	pNode : POINTER TO Node_F_VN_InvertMatrix3x3;
END_VAR
pNode := __NEW(Node_F_VN_InvertMatrix3x3);
Clone := pNode^;
END_METHOD

METHOD PROTECTED OnExecute
hresult.Value := F_VN_InvertMatrix3x3(
	aSrcMatrix := aSrcMatrix.Value,
    aInvertedMatrix := aInvertedMatrix.Value,
	hrPrev:= hrPrev.Value);
END_METHOD

METHOD PUBLIC PreExecutionCheck
VAR_INPUT
	Check : I_PreExecutionChecks;
END_VAR
END_METHOD

END_FUNCTION_BLOCK

// Nodes/Miscellaneous/Node_F_VN_LineIntersectionPoint
{attribute 'linkalways'} 
{attribute 'no_explicit_call' := 'This FB is a CLASS and must be accessed using methods or properties'}
{attribute 'enable_dynamic_creation'}
FUNCTION_BLOCK Node_F_VN_LineIntersectionPoint EXTENDS VisionNode
VAR
    aLine1 : _TcVnVector4_LREAL;
    aLine2 : _TcVnVector4_LREAL;
    aIntersecPoint : _TcVnPoint2_REAL;
    hrPrev : _HRESULT(S_OK);
	hresult : _HRESULT(S_OK);
END_VAR

METHOD FB_init : BOOL
VAR_INPUT
	bInitRetains : BOOL; // if TRUE, the retain variables are initialized (warm start / cold start)
	bInCopyCode : BOOL;  // if TRUE, the instance afterwards gets moved into the copy code (online change)
END_VAR
AddInput('aLine1', aLine1);
AddInput('aLine2', aLine2);
AddInput('hrPrev', hrPrev);
AddOutput('aIntersecPoint', aIntersecPoint);
AddOutput('hresult',hresult);
END_METHOD

METHOD PUBLIC  Clone : I_Node
VAR
	pNode : POINTER TO Node_F_VN_LineIntersectionPoint;
END_VAR
pNode := __NEW(Node_F_VN_LineIntersectionPoint);
Clone := pNode^;
END_METHOD

METHOD PROTECTED OnExecute
hresult.Value := F_VN_LineIntersectionPoint(
	aLine1 := aLine1.Value,
    aLine2 := aLine2.Value,
    aIntersecPoint := aIntersecPoint.Value,
	hrPrev:= hrPrev.Value);
END_METHOD

METHOD PUBLIC PreExecutionCheck
VAR_INPUT
	Check : I_PreExecutionChecks;
END_VAR
END_METHOD

END_FUNCTION_BLOCK

// Nodes/Miscellaneous/Node_F_VN_LineIntersectionPointAndAngle
{attribute 'linkalways'} 
{attribute 'no_explicit_call' := 'This FB is a CLASS and must be accessed using methods or properties'}
{attribute 'enable_dynamic_creation'}
FUNCTION_BLOCK Node_F_VN_LineIntersectionPointAndAngle EXTENDS VisionNode
VAR
    aLine1 : _TcVnVector4_LREAL;
    aLine2 : _TcVnVector4_LREAL;
    aIntersecPoint : _TcVnPoint2_REAL;
    fAngle : _REAL(0.0);
    bAngleInDegrees : _BOOL(FALSE);
    hrPrev : _HRESULT(S_OK);
	hresult : _HRESULT(S_OK);
END_VAR

METHOD FB_init : BOOL
VAR_INPUT
	bInitRetains : BOOL; // if TRUE, the retain variables are initialized (warm start / cold start)
	bInCopyCode : BOOL;  // if TRUE, the instance afterwards gets moved into the copy code (online change)
END_VAR
AddInput('aLine1', aLine1);
AddInput('aLine2', aLine2);
AddParameter('bAngleInDegrees', bAngleInDegrees);
AddInput('hrPrev', hrPrev);
AddOutput('aIntersecPoint', aIntersecPoint);
AddOutput('fAngle', fAngle);
AddOutput('hresult',hresult);
END_METHOD

METHOD PUBLIC  Clone : I_Node
VAR
	pNode : POINTER TO Node_F_VN_LineIntersectionPointAndAngle;
END_VAR
pNode := __NEW(Node_F_VN_LineIntersectionPointAndAngle);
Clone := pNode^;
END_METHOD

METHOD PROTECTED OnExecute
hresult.Value := F_VN_LineIntersectionPointAndAngle(
	aLine1 := aLine1.Value,
    aLine2 := aLine2.Value,
    aIntersecPoint := aIntersecPoint.Value,
    fAngle := fAngle.Value,
    bAngleInDegrees := bAngleInDegrees.Value,
	hrPrev:= hrPrev.Value);
END_METHOD

METHOD PUBLIC PreExecutionCheck
VAR_INPUT
	Check : I_PreExecutionChecks;
END_VAR
END_METHOD

END_FUNCTION_BLOCK

// Nodes/Miscellaneous/Node_F_VN_OrthogonalVector_TcVnVector2_DINT
{attribute 'linkalways'} 
{attribute 'no_explicit_call' := 'This FB is a CLASS and must be accessed using methods or properties'}
{attribute 'enable_dynamic_creation'}
FUNCTION_BLOCK Node_F_VN_OrthogonalVector_TcVnVector2_DINT EXTENDS VisionNode
VAR
    aSrc : _TcVnVector2_DINT;
    aOrthogonal : _TcVnVector2_LREAL;
    bNormalize : _BOOL(FALSE);
    hrPrev : _HRESULT(S_OK);
	hresult : _HRESULT(S_OK);
END_VAR

METHOD FB_init : BOOL
VAR_INPUT
	bInitRetains : BOOL; // if TRUE, the retain variables are initialized (warm start / cold start)
	bInCopyCode : BOOL;  // if TRUE, the instance afterwards gets moved into the copy code (online change)
END_VAR
AddInput('aSrc', aSrc);
AddParameter('bNormalize', bNormalize);
AddInput('hrPrev', hrPrev);
AddOutput('aOrthogonal', aOrthogonal);
AddOutput('hresult',hresult);
END_METHOD

METHOD PUBLIC  Clone : I_Node
VAR
	pNode : POINTER TO Node_F_VN_OrthogonalVector_TcVnVector2_DINT;
END_VAR
pNode := __NEW(Node_F_VN_OrthogonalVector_TcVnVector2_DINT);
Clone := pNode^;
END_METHOD

METHOD PROTECTED OnExecute
hresult.Value := F_VN_OrthogonalVector_TcVnVector2_DINT(
    aSrc := aSrc.Value,
    aOrthogonal := aOrthogonal.Value,
    bNormalize := bNormalize.Value,
	hrPrev:= hrPrev.Value);
END_METHOD

METHOD PUBLIC PreExecutionCheck
VAR_INPUT
	Check : I_PreExecutionChecks;
END_VAR
END_METHOD

END_FUNCTION_BLOCK

// Nodes/Miscellaneous/Node_F_VN_OrthogonalVector_TcVnVector2_LREAL
{attribute 'linkalways'} 
{attribute 'no_explicit_call' := 'This FB is a CLASS and must be accessed using methods or properties'}
{attribute 'enable_dynamic_creation'}
FUNCTION_BLOCK Node_F_VN_OrthogonalVector_TcVnVector2_LREAL EXTENDS VisionNode
VAR
    aSrc : _TcVnVector2_LREAL;
    aOrthogonal : _TcVnVector2_LREAL;
    bNormalize : _BOOL(FALSE);
    hrPrev : _HRESULT(S_OK);
	hresult : _HRESULT(S_OK);
END_VAR

METHOD FB_init : BOOL
VAR_INPUT
	bInitRetains : BOOL; // if TRUE, the retain variables are initialized (warm start / cold start)
	bInCopyCode : BOOL;  // if TRUE, the instance afterwards gets moved into the copy code (online change)
END_VAR
AddInput('aSrc', aSrc);
AddParameter('bNormalize', bNormalize);
AddInput('hrPrev', hrPrev);
AddOutput('aOrthogonal', aOrthogonal);
AddOutput('hresult',hresult);
END_METHOD

METHOD PUBLIC  Clone : I_Node
VAR
	pNode : POINTER TO Node_F_VN_OrthogonalVector_TcVnVector2_LREAL;
END_VAR
pNode := __NEW(Node_F_VN_OrthogonalVector_TcVnVector2_LREAL);
Clone := pNode^;
END_METHOD

METHOD PROTECTED OnExecute
hresult.Value := F_VN_OrthogonalVector_TcVnVector2_LREAL(
    aSrc := aSrc.Value,
    aOrthogonal := aOrthogonal.Value,
    bNormalize := bNormalize.Value,
	hrPrev:= hrPrev.Value);
END_METHOD

METHOD PUBLIC PreExecutionCheck
VAR_INPUT
	Check : I_PreExecutionChecks;
END_VAR
END_METHOD

END_FUNCTION_BLOCK

// Nodes/Miscellaneous/Node_F_VN_OrthogonalVector_TcVnVector2_REAL
{attribute 'linkalways'} 
{attribute 'no_explicit_call' := 'This FB is a CLASS and must be accessed using methods or properties'}
{attribute 'enable_dynamic_creation'}
FUNCTION_BLOCK Node_F_VN_OrthogonalVector_TcVnVector2_REAL EXTENDS VisionNode
VAR
    aSrc : _TcVnVector2_REAL;
    aOrthogonal : _TcVnVector2_REAL;
    bNormalize : _BOOL(FALSE);
    hrPrev : _HRESULT(S_OK);
	hresult : _HRESULT(S_OK);
END_VAR

METHOD FB_init : BOOL
VAR_INPUT
	bInitRetains : BOOL; // if TRUE, the retain variables are initialized (warm start / cold start)
	bInCopyCode : BOOL;  // if TRUE, the instance afterwards gets moved into the copy code (online change)
END_VAR
AddInput('aSrc', aSrc);
AddParameter('bNormalize', bNormalize);
AddInput('hrPrev', hrPrev);
AddOutput('aOrthogonal', aOrthogonal);
AddOutput('hresult',hresult);
END_METHOD

METHOD PUBLIC  Clone : I_Node
VAR
	pNode : POINTER TO Node_F_VN_OrthogonalVector_TcVnVector2_REAL;
END_VAR
pNode := __NEW(Node_F_VN_OrthogonalVector_TcVnVector2_REAL);
Clone := pNode^;
END_METHOD

METHOD PROTECTED OnExecute
hresult.Value := F_VN_OrthogonalVector_TcVnVector2_REAL(
    aSrc := aSrc.Value,
    aOrthogonal := aOrthogonal.Value,
    bNormalize := bNormalize.Value,
	hrPrev:= hrPrev.Value);
END_METHOD

METHOD PUBLIC PreExecutionCheck
VAR_INPUT
	Check : I_PreExecutionChecks;
END_VAR
END_METHOD

END_FUNCTION_BLOCK

// Nodes/Miscellaneous/Node_F_VN_PointToLineDistance_TcVnPoint2_DINT
{attribute 'linkalways'} 
{attribute 'no_explicit_call' := 'This FB is a CLASS and must be accessed using methods or properties'}
{attribute 'enable_dynamic_creation'}
FUNCTION_BLOCK Node_F_VN_PointToLineDistance_TcVnPoint2_DINT EXTENDS VisionNode
VAR
    aPoint : _TcVnPoint2_DINT;
    aLinePoint1 : _TcVnPoint2_DINT;
    aLinePoint2 : _TcVnPoint2_DINT;
    fDistance : _LREAL(0.0);
    hrPrev : _HRESULT(S_OK);
	hresult : _HRESULT(S_OK);
END_VAR

METHOD FB_init : BOOL
VAR_INPUT
	bInitRetains : BOOL; // if TRUE, the retain variables are initialized (warm start / cold start)
	bInCopyCode : BOOL;  // if TRUE, the instance afterwards gets moved into the copy code (online change)
END_VAR
AddInput('aPoint', aPoint);
AddInput('aLinePoint1', aLinePoint1);
AddInput('aLinePoint2', aLinePoint2);
AddInput('hrPrev', hrPrev);
AddOutput('fDistance', fDistance);
AddOutput('hresult',hresult);
END_METHOD

METHOD PUBLIC  Clone : I_Node
VAR
	pNode : POINTER TO Node_F_VN_PointToLineDistance_TcVnPoint2_DINT;
END_VAR
pNode := __NEW(Node_F_VN_PointToLineDistance_TcVnPoint2_DINT);
Clone := pNode^;
END_METHOD

METHOD PROTECTED OnExecute
hresult.Value := F_VN_PointToLineDistance_TcVnPoint2_DINT(
	aPoint := aPoint.Value,
    aLinePoint1 := aLinePoint1.Value,
    aLinePoint2 := aLinePoint2.Value,
    fDistance := fDistance.Value,
	hrPrev:= hrPrev.Value);
END_METHOD

METHOD PUBLIC PreExecutionCheck
VAR_INPUT
	Check : I_PreExecutionChecks;
END_VAR
END_METHOD

END_FUNCTION_BLOCK

// Nodes/Miscellaneous/Node_F_VN_PointToLineDistance_TcVnPoint2_LREAL
{attribute 'linkalways'} 
{attribute 'no_explicit_call' := 'This FB is a CLASS and must be accessed using methods or properties'}
{attribute 'enable_dynamic_creation'}
FUNCTION_BLOCK Node_F_VN_PointToLineDistance_TcVnPoint2_LREAL EXTENDS VisionNode
VAR
    aPoint : _TcVnPoint2_LREAL;
    aLinePoint1 : _TcVnPoint2_LREAL;
    aLinePoint2 : _TcVnPoint2_LREAL;
    fDistance : _LREAL(0.0);
    hrPrev : _HRESULT(S_OK);
	hresult : _HRESULT(S_OK);
END_VAR

METHOD FB_init : BOOL
VAR_INPUT
	bInitRetains : BOOL; // if TRUE, the retain variables are initialized (warm start / cold start)
	bInCopyCode : BOOL;  // if TRUE, the instance afterwards gets moved into the copy code (online change)
END_VAR
AddInput('aPoint', aPoint);
AddInput('aLinePoint1', aLinePoint1);
AddInput('aLinePoint2', aLinePoint2);
AddInput('hrPrev', hrPrev);
AddOutput('fDistance', fDistance);
AddOutput('hresult',hresult);
END_METHOD

METHOD PUBLIC  Clone : I_Node
VAR
	pNode : POINTER TO Node_F_VN_PointToLineDistance_TcVnPoint2_LREAL;
END_VAR
pNode := __NEW(Node_F_VN_PointToLineDistance_TcVnPoint2_LREAL);
Clone := pNode^;
END_METHOD

METHOD PROTECTED OnExecute
hresult.Value := F_VN_PointToLineDistance_TcVnPoint2_LREAL(
	aPoint := aPoint.Value,
    aLinePoint1 := aLinePoint1.Value,
    aLinePoint2 := aLinePoint2.Value,
    fDistance := fDistance.Value,
	hrPrev:= hrPrev.Value);
END_METHOD

METHOD PUBLIC PreExecutionCheck
VAR_INPUT
	Check : I_PreExecutionChecks;
END_VAR
END_METHOD

END_FUNCTION_BLOCK

// Nodes/Miscellaneous/Node_F_VN_PointToLineDistance_TcVnPoint2_REAL
{attribute 'linkalways'} 
{attribute 'no_explicit_call' := 'This FB is a CLASS and must be accessed using methods or properties'}
{attribute 'enable_dynamic_creation'}
FUNCTION_BLOCK Node_F_VN_PointToLineDistance_TcVnPoint2_REAL EXTENDS VisionNode
VAR
    aPoint : _TcVnPoint2_REAL;
    aLinePoint1 : _TcVnPoint2_REAL;
    aLinePoint2 : _TcVnPoint2_REAL;
    fDistance : _LREAL(0.0);
    hrPrev : _HRESULT(S_OK);
	hresult : _HRESULT(S_OK);
END_VAR

METHOD FB_init : BOOL
VAR_INPUT
	bInitRetains : BOOL; // if TRUE, the retain variables are initialized (warm start / cold start)
	bInCopyCode : BOOL;  // if TRUE, the instance afterwards gets moved into the copy code (online change)
END_VAR
AddInput('aPoint', aPoint);
AddInput('aLinePoint1', aLinePoint1);
AddInput('aLinePoint2', aLinePoint2);
AddInput('hrPrev', hrPrev);
AddOutput('fDistance', fDistance);
AddOutput('hresult',hresult);
END_METHOD

METHOD PUBLIC  Clone : I_Node
VAR
	pNode : POINTER TO Node_F_VN_PointToLineDistance_TcVnPoint2_REAL;
END_VAR
pNode := __NEW(Node_F_VN_PointToLineDistance_TcVnPoint2_REAL);
Clone := pNode^;
END_METHOD

METHOD PROTECTED OnExecute
hresult.Value := F_VN_PointToLineDistance_TcVnPoint2_REAL(
	aPoint := aPoint.Value,
    aLinePoint1 := aLinePoint1.Value,
    aLinePoint2 := aLinePoint2.Value,
    fDistance := fDistance.Value,
	hrPrev:= hrPrev.Value);
END_METHOD

METHOD PUBLIC PreExecutionCheck
VAR_INPUT
	Check : I_PreExecutionChecks;
END_VAR
END_METHOD

END_FUNCTION_BLOCK

// Nodes/Miscellaneous/Node_F_VN_PointToPointDirection_TcVnPoint2_DINT
{attribute 'linkalways'} 
{attribute 'no_explicit_call' := 'This FB is a CLASS and must be accessed using methods or properties'}
{attribute 'enable_dynamic_creation'}
FUNCTION_BLOCK Node_F_VN_PointToPointDirection_TcVnPoint2_DINT EXTENDS VisionNode
VAR
    aPoint1 : _TcVnPoint2_DINT;
    aPoint2 : _TcVnPoint2_DINT;
    aDirection : _TcVnVector2_LREAL;
    bNormalize : _BOOL(FALSE);
    hrPrev : _HRESULT(S_OK);
	hresult : _HRESULT(S_OK);
END_VAR

